// TIA Portal V18 export
// export: Created 2026-01-09T11:31:54.3850951Z, ExportSetting WithDefaults, DisplayName Totally Integrated Automation Portal, DisplayVersion V18 Update 5, DisplayName TIA Portal Openness, DisplayVersion V18 Update 5, DisplayName TIA Portal Teamcenter Gateway, DisplayVersion V18, DisplayName TIA Portal Version Control Interface, DisplayVersion V18, DisplayName SINAMICS Startdrive Advanced, DisplayVersion V18 SP2 Update 1, DisplayName SINAMICS Startdrive G110M, G120, G120C, G120D, G120P, G115D, DisplayVersion V18 SP2 Update 1, DisplayName SINAMICS Startdrive G130, G150, S120, S150, SINAMICS MV, S210, G220, S200, DisplayVersion V18 SP2 Update 1, DisplayName STEP 7 Professional, DisplayVersion V18 Update 5, DisplayName STEP 7 Safety, DisplayVersion V18, DisplayName WinCC Professional, DisplayVersion V18 Update 5
TagTable "ST350_CylinderV2"
  STxxxCylinder001 : fpCylinder V 0.0.19  (%DB1020.DBX0.0, CPU S71500-2PN_TP700, 1 s)
    TagStructureMember "InWP"  LogicalAddress=%DB1020.DBX0.3
    TagStructureMember "InHP"  LogicalAddress=%DB1020.DBX0.4
    TagStructureMember "ValveType"  LogicalAddress=%DB1020.DBX0.5
    TagStructureMember "ManualToWP"  LogicalAddress=%DB1020.DBX6.0
    TagStructureMember "ManualToHP"  LogicalAddress=%DB1020.DBX6.1
    TagStructureMember "GoWorkTime"  LogicalAddress=%DB1020.DBW8
    TagStructureMember "GoHomeTime"  LogicalAddress=%DB1020.DBW10
    TagStructureMember "oGoWP"  LogicalAddress=%DB1020.DBX20.0
    TagStructureMember "oGoHP"  LogicalAddress=%DB1020.DBX20.1
    TagStructureMember "oGoWPBTActive"  LogicalAddress=%DB1020.DBX20.2
    TagStructureMember "oGoHPBTActive"  LogicalAddress=%DB1020.DBX20.3
    TagStructureMember "CylinderNo"  LogicalAddress=%DB1020.DBB21
  STxxxCylinder002 : fpCylinder V 0.0.19  (%DB1020.DBX22.0, CPU S71500-2PN_TP700, 1 s)
    TagStructureMember "InWP"  LogicalAddress=%DB1020.DBX22.3
    TagStructureMember "InHP"  LogicalAddress=%DB1020.DBX22.4
    TagStructureMember "ValveType"  LogicalAddress=%DB1020.DBX22.5
    TagStructureMember "ManualToWP"  LogicalAddress=%DB1020.DBX28.0
    TagStructureMember "ManualToHP"  LogicalAddress=%DB1020.DBX28.1
    TagStructureMember "GoWorkTime"  LogicalAddress=%DB1020.DBW30
    TagStructureMember "GoHomeTime"  LogicalAddress=%DB1020.DBW32
    TagStructureMember "oGoWP"  LogicalAddress=%DB1020.DBX42.0
    TagStructureMember "oGoHP"  LogicalAddress=%DB1020.DBX42.1
    TagStructureMember "oGoWPBTActive"  LogicalAddress=%DB1020.DBX42.2
    TagStructureMember "oGoHPBTActive"  LogicalAddress=%DB1020.DBX42.3
    TagStructureMember "CylinderNo"  LogicalAddress=%DB1020.DBB43
  STxxxCylinder003 : fpCylinder V 0.0.19  (%DB1020.DBX44.0, CPU S71500-2PN_TP700, 1 s)
    TagStructureMember "InWP"  LogicalAddress=%DB1020.DBX44.3
    TagStructureMember "InHP"  LogicalAddress=%DB1020.DBX44.4
    TagStructureMember "ValveType"  LogicalAddress=%DB1020.DBX44.5
    TagStructureMember "ManualToWP"  LogicalAddress=%DB1020.DBX50.0
    TagStructureMember "ManualToHP"  LogicalAddress=%DB1020.DBX50.1
    TagStructureMember "GoWorkTime"  LogicalAddress=%DB1020.DBW52
    TagStructureMember "GoHomeTime"  LogicalAddress=%DB1020.DBW54
    TagStructureMember "oGoWP"  LogicalAddress=%DB1020.DBX64.0
    TagStructureMember "oGoHP"  LogicalAddress=%DB1020.DBX64.1
    TagStructureMember "oGoWPBTActive"  LogicalAddress=%DB1020.DBX64.2
    TagStructureMember "oGoHPBTActive"  LogicalAddress=%DB1020.DBX64.3
    TagStructureMember "CylinderNo"  LogicalAddress=%DB1020.DBB65
  STxxxCylinder004 : fpCylinder V 0.0.19  (%DB1020.DBX66.0, CPU S71500-2PN_TP700, 1 s)
    TagStructureMember "InWP"  LogicalAddress=%DB1020.DBX66.3
    TagStructureMember "InHP"  LogicalAddress=%DB1020.DBX66.4
    TagStructureMember "ValveType"  LogicalAddress=%DB1020.DBX66.5
    TagStructureMember "ManualToWP"  LogicalAddress=%DB1020.DBX72.0
    TagStructureMember "ManualToHP"  LogicalAddress=%DB1020.DBX72.1
    TagStructureMember "GoWorkTime"  LogicalAddress=%DB1020.DBW74
    TagStructureMember "GoHomeTime"  LogicalAddress=%DB1020.DBW76
    TagStructureMember "oGoWP"  LogicalAddress=%DB1020.DBX86.0
    TagStructureMember "oGoHP"  LogicalAddress=%DB1020.DBX86.1
    TagStructureMember "oGoWPBTActive"  LogicalAddress=%DB1020.DBX86.2
    TagStructureMember "oGoHPBTActive"  LogicalAddress=%DB1020.DBX86.3
    TagStructureMember "CylinderNo"  LogicalAddress=%DB1020.DBB87
  STxxxCylinder005 : fpCylinder V 0.0.19  (%DB1020.DBX88.0, CPU S71500-2PN_TP700, 1 s)
    TagStructureMember "InWP"  LogicalAddress=%DB1020.DBX88.3
    TagStructureMember "InHP"  LogicalAddress=%DB1020.DBX88.4
    TagStructureMember "ValveType"  LogicalAddress=%DB1020.DBX88.5
    TagStructureMember "ManualToWP"  LogicalAddress=%DB1020.DBX94.0
    TagStructureMember "ManualToHP"  LogicalAddress=%DB1020.DBX94.1
    TagStructureMember "GoWorkTime"  LogicalAddress=%DB1020.DBW96
    TagStructureMember "GoHomeTime"  LogicalAddress=%DB1020.DBW98
    TagStructureMember "oGoWP"  LogicalAddress=%DB1020.DBX108.0
    TagStructureMember "oGoHP"  LogicalAddress=%DB1020.DBX108.1
    TagStructureMember "oGoWPBTActive"  LogicalAddress=%DB1020.DBX108.2
    TagStructureMember "oGoHPBTActive"  LogicalAddress=%DB1020.DBX108.3
    TagStructureMember "CylinderNo"  LogicalAddress=%DB1020.DBB109
  STxxxCylinder006 : fpCylinder V 0.0.19  (%DB1020.DBX110.0, CPU S71500-2PN_TP700, 1 s)
    TagStructureMember "InWP"  LogicalAddress=%DB1020.DBX110.3
    TagStructureMember "InHP"  LogicalAddress=%DB1020.DBX110.4
    TagStructureMember "ValveType"  LogicalAddress=%DB1020.DBX110.5
    TagStructureMember "ManualToWP"  LogicalAddress=%DB1020.DBX116.0
    TagStructureMember "ManualToHP"  LogicalAddress=%DB1020.DBX116.1
    TagStructureMember "GoWorkTime"  LogicalAddress=%DB1020.DBW118
    TagStructureMember "GoHomeTime"  LogicalAddress=%DB1020.DBW120
    TagStructureMember "oGoWP"  LogicalAddress=%DB1020.DBX130.0
    TagStructureMember "oGoHP"  LogicalAddress=%DB1020.DBX130.1
    TagStructureMember "oGoWPBTActive"  LogicalAddress=%DB1020.DBX130.2
    TagStructureMember "oGoHPBTActive"  LogicalAddress=%DB1020.DBX130.3
    TagStructureMember "CylinderNo"  LogicalAddress=%DB1020.DBB131
  STxxxCylinder007 : fpCylinder V 0.0.19  (%DB1020.DBX132.0, CPU S71500-2PN_TP700, 1 s)
    TagStructureMember "InWP"  LogicalAddress=%DB1020.DBX132.3
    TagStructureMember "InHP"  LogicalAddress=%DB1020.DBX132.4
    TagStructureMember "ValveType"  LogicalAddress=%DB1020.DBX132.5
    TagStructureMember "ManualToWP"  LogicalAddress=%DB1020.DBX138.0
    TagStructureMember "ManualToHP"  LogicalAddress=%DB1020.DBX138.1
    TagStructureMember "GoWorkTime"  LogicalAddress=%DB1020.DBW140
    TagStructureMember "GoHomeTime"  LogicalAddress=%DB1020.DBW142
    TagStructureMember "oGoWP"  LogicalAddress=%DB1020.DBX152.0
    TagStructureMember "oGoHP"  LogicalAddress=%DB1020.DBX152.1
    TagStructureMember "oGoWPBTActive"  LogicalAddress=%DB1020.DBX152.2
    TagStructureMember "oGoHPBTActive"  LogicalAddress=%DB1020.DBX152.3
    TagStructureMember "CylinderNo"  LogicalAddress=%DB1020.DBB153
  STxxxCylinder008 : fpCylinder V 0.0.19  (%DB1020.DBX154.0, CPU S71500-2PN_TP700, 1 s)
    TagStructureMember "InWP"  LogicalAddress=%DB1020.DBX154.3
    TagStructureMember "InHP"  LogicalAddress=%DB1020.DBX154.4
    TagStructureMember "ValveType"  LogicalAddress=%DB1020.DBX154.5
    TagStructureMember "ManualToWP"  LogicalAddress=%DB1020.DBX160.0
    TagStructureMember "ManualToHP"  LogicalAddress=%DB1020.DBX160.1
    TagStructureMember "GoWorkTime"  LogicalAddress=%DB1020.DBW162
    TagStructureMember "GoHomeTime"  LogicalAddress=%DB1020.DBW164
    TagStructureMember "oGoWP"  LogicalAddress=%DB1020.DBX174.0
    TagStructureMember "oGoHP"  LogicalAddress=%DB1020.DBX174.1
    TagStructureMember "oGoWPBTActive"  LogicalAddress=%DB1020.DBX174.2
    TagStructureMember "oGoHPBTActive"  LogicalAddress=%DB1020.DBX174.3
    TagStructureMember "CylinderNo"  LogicalAddress=%DB1020.DBB175
  STxxxCylinder009 : fpCylinder V 0.0.19  (%DB1020.DBX176.0, CPU S71500-2PN_TP700, 1 s)
    TagStructureMember "InWP"  LogicalAddress=%DB1020.DBX176.3
    TagStructureMember "InHP"  LogicalAddress=%DB1020.DBX176.4
    TagStructureMember "ValveType"  LogicalAddress=%DB1020.DBX176.5
    TagStructureMember "ManualToWP"  LogicalAddress=%DB1020.DBX182.0
    TagStructureMember "ManualToHP"  LogicalAddress=%DB1020.DBX182.1
    TagStructureMember "GoWorkTime"  LogicalAddress=%DB1020.DBW184
    TagStructureMember "GoHomeTime"  LogicalAddress=%DB1020.DBW186
    TagStructureMember "oGoWP"  LogicalAddress=%DB1020.DBX196.0
    TagStructureMember "oGoHP"  LogicalAddress=%DB1020.DBX196.1
    TagStructureMember "oGoWPBTActive"  LogicalAddress=%DB1020.DBX196.2
    TagStructureMember "oGoHPBTActive"  LogicalAddress=%DB1020.DBX196.3
    TagStructureMember "CylinderNo"  LogicalAddress=%DB1020.DBB197
  STxxxCylinder010 : fpCylinder V 0.0.19  (%DB1020.DBX198.0, CPU S71500-2PN_TP700, 1 s)
    TagStructureMember "InWP"  LogicalAddress=%DB1020.DBX198.3
    TagStructureMember "InHP"  LogicalAddress=%DB1020.DBX198.4
    TagStructureMember "ValveType"  LogicalAddress=%DB1020.DBX198.5
    TagStructureMember "ManualToWP"  LogicalAddress=%DB1020.DBX204.0
    TagStructureMember "ManualToHP"  LogicalAddress=%DB1020.DBX204.1
    TagStructureMember "GoWorkTime"  LogicalAddress=%DB1020.DBW206
    TagStructureMember "GoHomeTime"  LogicalAddress=%DB1020.DBW208
    TagStructureMember "oGoWP"  LogicalAddress=%DB1020.DBX218.0
    TagStructureMember "oGoHP"  LogicalAddress=%DB1020.DBX218.1
    TagStructureMember "oGoWPBTActive"  LogicalAddress=%DB1020.DBX218.2
    TagStructureMember "oGoHPBTActive"  LogicalAddress=%DB1020.DBX218.3
    TagStructureMember "CylinderNo"  LogicalAddress=%DB1020.DBB219
  STxxxCylinder011 : fpCylinder V 0.0.19  (%DB1020.DBX220.0, CPU S71500-2PN_TP700, 1 s)
    TagStructureMember "InWP"  LogicalAddress=%DB1020.DBX220.3
    TagStructureMember "InHP"  LogicalAddress=%DB1020.DBX220.4
    TagStructureMember "ValveType"  LogicalAddress=%DB1020.DBX220.5
    TagStructureMember "ManualToWP"  LogicalAddress=%DB1020.DBX226.0
    TagStructureMember "ManualToHP"  LogicalAddress=%DB1020.DBX226.1
    TagStructureMember "GoWorkTime"  LogicalAddress=%DB1020.DBW228
    TagStructureMember "GoHomeTime"  LogicalAddress=%DB1020.DBW230
    TagStructureMember "oGoWP"  LogicalAddress=%DB1020.DBX240.0
    TagStructureMember "oGoHP"  LogicalAddress=%DB1020.DBX240.1
    TagStructureMember "oGoWPBTActive"  LogicalAddress=%DB1020.DBX240.2
    TagStructureMember "oGoHPBTActive"  LogicalAddress=%DB1020.DBX240.3
    TagStructureMember "CylinderNo"  LogicalAddress=%DB1020.DBB241
  STxxxCylinder012 : fpCylinder V 0.0.19  (%DB1020.DBX242.0, CPU S71500-2PN_TP700, 1 s)
    TagStructureMember "InWP"  LogicalAddress=%DB1020.DBX242.3
    TagStructureMember "InHP"  LogicalAddress=%DB1020.DBX242.4
    TagStructureMember "ValveType"  LogicalAddress=%DB1020.DBX242.5
    TagStructureMember "ManualToWP"  LogicalAddress=%DB1020.DBX248.0
    TagStructureMember "ManualToHP"  LogicalAddress=%DB1020.DBX248.1
    TagStructureMember "GoWorkTime"  LogicalAddress=%DB1020.DBW250
    TagStructureMember "GoHomeTime"  LogicalAddress=%DB1020.DBW252
    TagStructureMember "oGoWP"  LogicalAddress=%DB1020.DBX262.0
    TagStructureMember "oGoHP"  LogicalAddress=%DB1020.DBX262.1
    TagStructureMember "oGoWPBTActive"  LogicalAddress=%DB1020.DBX262.2
    TagStructureMember "oGoHPBTActive"  LogicalAddress=%DB1020.DBX262.3
    TagStructureMember "CylinderNo"  LogicalAddress=%DB1020.DBB263
  STxxxCylinder013 : fpCylinder V 0.0.19  (%DB1020.DBX264.0, CPU S71500-2PN_TP700, 1 s)
    TagStructureMember "InWP"  LogicalAddress=%DB1020.DBX264.3
    TagStructureMember "InHP"  LogicalAddress=%DB1020.DBX264.4
    TagStructureMember "ValveType"  LogicalAddress=%DB1020.DBX264.5
    TagStructureMember "ManualToWP"  LogicalAddress=%DB1020.DBX270.0
    TagStructureMember "ManualToHP"  LogicalAddress=%DB1020.DBX270.1
    TagStructureMember "GoWorkTime"  LogicalAddress=%DB1020.DBW272
    TagStructureMember "GoHomeTime"  LogicalAddress=%DB1020.DBW274
    TagStructureMember "oGoWP"  LogicalAddress=%DB1020.DBX284.0
    TagStructureMember "oGoHP"  LogicalAddress=%DB1020.DBX284.1
    TagStructureMember "oGoWPBTActive"  LogicalAddress=%DB1020.DBX284.2
    TagStructureMember "oGoHPBTActive"  LogicalAddress=%DB1020.DBX284.3
    TagStructureMember "CylinderNo"  LogicalAddress=%DB1020.DBB285
  STxxxCylinder014 : fpCylinder V 0.0.19  (%DB1020.DBX286.0, CPU S71500-2PN_TP700, 1 s)
    TagStructureMember "InWP"  LogicalAddress=%DB1020.DBX286.3
    TagStructureMember "InHP"  LogicalAddress=%DB1020.DBX286.4
    TagStructureMember "ValveType"  LogicalAddress=%DB1020.DBX286.5
    TagStructureMember "ManualToWP"  LogicalAddress=%DB1020.DBX292.0
    TagStructureMember "ManualToHP"  LogicalAddress=%DB1020.DBX292.1
    TagStructureMember "GoWorkTime"  LogicalAddress=%DB1020.DBW294
    TagStructureMember "GoHomeTime"  LogicalAddress=%DB1020.DBW296
    TagStructureMember "oGoWP"  LogicalAddress=%DB1020.DBX306.0
    TagStructureMember "oGoHP"  LogicalAddress=%DB1020.DBX306.1
    TagStructureMember "oGoWPBTActive"  LogicalAddress=%DB1020.DBX306.2
    TagStructureMember "oGoHPBTActive"  LogicalAddress=%DB1020.DBX306.3
    TagStructureMember "CylinderNo"  LogicalAddress=%DB1020.DBB307
  STxxxCylinder015 : fpCylinder V 0.0.19  (%DB1020.DBX308.0, CPU S71500-2PN_TP700, 1 s)
    TagStructureMember "InWP"  LogicalAddress=%DB1020.DBX308.3
    TagStructureMember "InHP"  LogicalAddress=%DB1020.DBX308.4
    TagStructureMember "ValveType"  LogicalAddress=%DB1020.DBX308.5
    TagStructureMember "ManualToWP"  LogicalAddress=%DB1020.DBX314.0
    TagStructureMember "ManualToHP"  LogicalAddress=%DB1020.DBX314.1
    TagStructureMember "GoWorkTime"  LogicalAddress=%DB1020.DBW316
    TagStructureMember "GoHomeTime"  LogicalAddress=%DB1020.DBW318
    TagStructureMember "oGoWP"  LogicalAddress=%DB1020.DBX328.0
    TagStructureMember "oGoHP"  LogicalAddress=%DB1020.DBX328.1
    TagStructureMember "oGoWPBTActive"  LogicalAddress=%DB1020.DBX328.2
    TagStructureMember "oGoHPBTActive"  LogicalAddress=%DB1020.DBX328.3
    TagStructureMember "CylinderNo"  LogicalAddress=%DB1020.DBB329
  STxxxCylinder016 : fpCylinder V 0.0.19  (%DB1020.DBX330.0, CPU S71500-2PN_TP700, 1 s)
    TagStructureMember "InWP"  LogicalAddress=%DB1020.DBX330.3
    TagStructureMember "InHP"  LogicalAddress=%DB1020.DBX330.4
    TagStructureMember "ValveType"  LogicalAddress=%DB1020.DBX330.5
    TagStructureMember "ManualToWP"  LogicalAddress=%DB1020.DBX336.0
    TagStructureMember "ManualToHP"  LogicalAddress=%DB1020.DBX336.1
    TagStructureMember "GoWorkTime"  LogicalAddress=%DB1020.DBW338
    TagStructureMember "GoHomeTime"  LogicalAddress=%DB1020.DBW340
    TagStructureMember "oGoWP"  LogicalAddress=%DB1020.DBX350.0
    TagStructureMember "oGoHP"  LogicalAddress=%DB1020.DBX350.1
    TagStructureMember "oGoWPBTActive"  LogicalAddress=%DB1020.DBX350.2
    TagStructureMember "oGoHPBTActive"  LogicalAddress=%DB1020.DBX350.3
    TagStructureMember "CylinderNo"  LogicalAddress=%DB1020.DBB351
  STxxxCylinder017 : fpCylinder V 0.0.19  (%DB1020.DBX352.0, CPU S71500-2PN_TP700, 1 s)
    TagStructureMember "InWP"  LogicalAddress=%DB1020.DBX352.3
    TagStructureMember "InHP"  LogicalAddress=%DB1020.DBX352.4
    TagStructureMember "ValveType"  LogicalAddress=%DB1020.DBX352.5
    TagStructureMember "ManualToWP"  LogicalAddress=%DB1020.DBX358.0
    TagStructureMember "ManualToHP"  LogicalAddress=%DB1020.DBX358.1
    TagStructureMember "GoWorkTime"  LogicalAddress=%DB1020.DBW360
    TagStructureMember "GoHomeTime"  LogicalAddress=%DB1020.DBW362
    TagStructureMember "oGoWP"  LogicalAddress=%DB1020.DBX372.0
    TagStructureMember "oGoHP"  LogicalAddress=%DB1020.DBX372.1
    TagStructureMember "oGoWPBTActive"  LogicalAddress=%DB1020.DBX372.2
    TagStructureMember "oGoHPBTActive"  LogicalAddress=%DB1020.DBX372.3
    TagStructureMember "CylinderNo"  LogicalAddress=%DB1020.DBB373
  STxxxCylinder018 : fpCylinder V 0.0.19  (%DB1020.DBX374.0, CPU S71500-2PN_TP700, 1 s)
    TagStructureMember "InWP"  LogicalAddress=%DB1020.DBX374.3
    TagStructureMember "InHP"  LogicalAddress=%DB1020.DBX374.4
    TagStructureMember "ValveType"  LogicalAddress=%DB1020.DBX374.5
    TagStructureMember "ManualToWP"  LogicalAddress=%DB1020.DBX380.0
    TagStructureMember "ManualToHP"  LogicalAddress=%DB1020.DBX380.1
    TagStructureMember "GoWorkTime"  LogicalAddress=%DB1020.DBW382
    TagStructureMember "GoHomeTime"  LogicalAddress=%DB1020.DBW384
    TagStructureMember "oGoWP"  LogicalAddress=%DB1020.DBX394.0
    TagStructureMember "oGoHP"  LogicalAddress=%DB1020.DBX394.1
    TagStructureMember "oGoWPBTActive"  LogicalAddress=%DB1020.DBX394.2
    TagStructureMember "oGoHPBTActive"  LogicalAddress=%DB1020.DBX394.3
    TagStructureMember "CylinderNo"  LogicalAddress=%DB1020.DBB395
  STxxxCylinder019 : fpCylinder V 0.0.19  (%DB1020.DBX396.0, CPU S71500-2PN_TP700, 1 s)
    TagStructureMember "InWP"  LogicalAddress=%DB1020.DBX396.3
    TagStructureMember "InHP"  LogicalAddress=%DB1020.DBX396.4
    TagStructureMember "ValveType"  LogicalAddress=%DB1020.DBX396.5
    TagStructureMember "ManualToWP"  LogicalAddress=%DB1020.DBX402.0
    TagStructureMember "ManualToHP"  LogicalAddress=%DB1020.DBX402.1
    TagStructureMember "GoWorkTime"  LogicalAddress=%DB1020.DBW404
    TagStructureMember "GoHomeTime"  LogicalAddress=%DB1020.DBW406
    TagStructureMember "oGoWP"  LogicalAddress=%DB1020.DBX416.0
    TagStructureMember "oGoHP"  LogicalAddress=%DB1020.DBX416.1
    TagStructureMember "oGoWPBTActive"  LogicalAddress=%DB1020.DBX416.2
    TagStructureMember "oGoHPBTActive"  LogicalAddress=%DB1020.DBX416.3
    TagStructureMember "CylinderNo"  LogicalAddress=%DB1020.DBB417
  STxxxCylinder020 : fpCylinder V 0.0.19  (%DB1020.DBX418.0, CPU S71500-2PN_TP700, 1 s)
    TagStructureMember "InWP"  LogicalAddress=%DB1020.DBX418.3
    TagStructureMember "InHP"  LogicalAddress=%DB1020.DBX418.4
    TagStructureMember "ValveType"  LogicalAddress=%DB1020.DBX418.5
    TagStructureMember "ManualToWP"  LogicalAddress=%DB1020.DBX424.0
    TagStructureMember "ManualToHP"  LogicalAddress=%DB1020.DBX424.1
    TagStructureMember "GoWorkTime"  LogicalAddress=%DB1020.DBW426
    TagStructureMember "GoHomeTime"  LogicalAddress=%DB1020.DBW428
    TagStructureMember "oGoWP"  LogicalAddress=%DB1020.DBX438.0
    TagStructureMember "oGoHP"  LogicalAddress=%DB1020.DBX438.1
    TagStructureMember "oGoWPBTActive"  LogicalAddress=%DB1020.DBX438.2
    TagStructureMember "oGoHPBTActive"  LogicalAddress=%DB1020.DBX438.3
    TagStructureMember "CylinderNo"  LogicalAddress=%DB1020.DBB439
  STxxxCylinder021 : fpCylinder V 0.0.19  (%DB1020.DBX440.0, CPU S71500-2PN_TP700, 1 s)
    TagStructureMember "InWP"  LogicalAddress=%DB1020.DBX440.3
    TagStructureMember "InHP"  LogicalAddress=%DB1020.DBX440.4
    TagStructureMember "ValveType"  LogicalAddress=%DB1020.DBX440.5
    TagStructureMember "ManualToWP"  LogicalAddress=%DB1020.DBX446.0
    TagStructureMember "ManualToHP"  LogicalAddress=%DB1020.DBX446.1
    TagStructureMember "GoWorkTime"  LogicalAddress=%DB1020.DBW448
    TagStructureMember "GoHomeTime"  LogicalAddress=%DB1020.DBW450
    TagStructureMember "oGoWP"  LogicalAddress=%DB1020.DBX460.0
    TagStructureMember "oGoHP"  LogicalAddress=%DB1020.DBX460.1
    TagStructureMember "oGoWPBTActive"  LogicalAddress=%DB1020.DBX460.2
    TagStructureMember "oGoHPBTActive"  LogicalAddress=%DB1020.DBX460.3
    TagStructureMember "CylinderNo"  LogicalAddress=%DB1020.DBB461
  STxxxCylinder022 : fpCylinder V 0.0.19  (%DB1020.DBX462.0, CPU S71500-2PN_TP700, 1 s)
    TagStructureMember "InWP"  LogicalAddress=%DB1020.DBX462.3
    TagStructureMember "InHP"  LogicalAddress=%DB1020.DBX462.4
    TagStructureMember "ValveType"  LogicalAddress=%DB1020.DBX462.5
    TagStructureMember "ManualToWP"  LogicalAddress=%DB1020.DBX468.0
    TagStructureMember "ManualToHP"  LogicalAddress=%DB1020.DBX468.1
    TagStructureMember "GoWorkTime"  LogicalAddress=%DB1020.DBW470
    TagStructureMember "GoHomeTime"  LogicalAddress=%DB1020.DBW472
    TagStructureMember "oGoWP"  LogicalAddress=%DB1020.DBX482.0
    TagStructureMember "oGoHP"  LogicalAddress=%DB1020.DBX482.1
    TagStructureMember "oGoWPBTActive"  LogicalAddress=%DB1020.DBX482.2
    TagStructureMember "oGoHPBTActive"  LogicalAddress=%DB1020.DBX482.3
    TagStructureMember "CylinderNo"  LogicalAddress=%DB1020.DBB483
  STxxxCylinder023 : fpCylinder V 0.0.19  (%DB1020.DBX484.0, CPU S71500-2PN_TP700, 1 s)
    TagStructureMember "InWP"  LogicalAddress=%DB1020.DBX484.3
    TagStructureMember "InHP"  LogicalAddress=%DB1020.DBX484.4
    TagStructureMember "ValveType"  LogicalAddress=%DB1020.DBX484.5
    TagStructureMember "ManualToWP"  LogicalAddress=%DB1020.DBX490.0
    TagStructureMember "ManualToHP"  LogicalAddress=%DB1020.DBX490.1
    TagStructureMember "GoWorkTime"  LogicalAddress=%DB1020.DBW492
    TagStructureMember "GoHomeTime"  LogicalAddress=%DB1020.DBW494
    TagStructureMember "oGoWP"  LogicalAddress=%DB1020.DBX504.0
    TagStructureMember "oGoHP"  LogicalAddress=%DB1020.DBX504.1
    TagStructureMember "oGoWPBTActive"  LogicalAddress=%DB1020.DBX504.2
    TagStructureMember "oGoHPBTActive"  LogicalAddress=%DB1020.DBX504.3
    TagStructureMember "CylinderNo"  LogicalAddress=%DB1020.DBB505
  STxxxCylinder024 : fpCylinder V 0.0.19  (%DB1020.DBX506.0, CPU S71500-2PN_TP700, 1 s)
    TagStructureMember "InWP"  LogicalAddress=%DB1020.DBX506.3
    TagStructureMember "InHP"  LogicalAddress=%DB1020.DBX506.4
    TagStructureMember "ValveType"  LogicalAddress=%DB1020.DBX506.5
    TagStructureMember "ManualToWP"  LogicalAddress=%DB1020.DBX512.0
    TagStructureMember "ManualToHP"  LogicalAddress=%DB1020.DBX512.1
    TagStructureMember "GoWorkTime"  LogicalAddress=%DB1020.DBW514
    TagStructureMember "GoHomeTime"  LogicalAddress=%DB1020.DBW516
    TagStructureMember "oGoWP"  LogicalAddress=%DB1020.DBX526.0
    TagStructureMember "oGoHP"  LogicalAddress=%DB1020.DBX526.1
    TagStructureMember "oGoWPBTActive"  LogicalAddress=%DB1020.DBX526.2
    TagStructureMember "oGoHPBTActive"  LogicalAddress=%DB1020.DBX526.3
    TagStructureMember "CylinderNo"  LogicalAddress=%DB1020.DBB527
  STxxxCylinder025 : fpCylinder V 0.0.19  (%DB1020.DBX528.0, CPU S71500-2PN_TP700, 1 s)
    TagStructureMember "InWP"  LogicalAddress=%DB1020.DBX528.3
    TagStructureMember "InHP"  LogicalAddress=%DB1020.DBX528.4
    TagStructureMember "ValveType"  LogicalAddress=%DB1020.DBX528.5
    TagStructureMember "ManualToWP"  LogicalAddress=%DB1020.DBX534.0
    TagStructureMember "ManualToHP"  LogicalAddress=%DB1020.DBX534.1
    TagStructureMember "GoWorkTime"  LogicalAddress=%DB1020.DBW536
    TagStructureMember "GoHomeTime"  LogicalAddress=%DB1020.DBW538
    TagStructureMember "oGoWP"  LogicalAddress=%DB1020.DBX548.0
    TagStructureMember "oGoHP"  LogicalAddress=%DB1020.DBX548.1
    TagStructureMember "oGoWPBTActive"  LogicalAddress=%DB1020.DBX548.2
    TagStructureMember "oGoHPBTActive"  LogicalAddress=%DB1020.DBX548.3
    TagStructureMember "CylinderNo"  LogicalAddress=%DB1020.DBB549
  STxxxCylinder026 : fpCylinder V 0.0.19  (%DB1020.DBX550.0, CPU S71500-2PN_TP700, 1 s)
    TagStructureMember "InWP"  LogicalAddress=%DB1020.DBX550.3
    TagStructureMember "InHP"  LogicalAddress=%DB1020.DBX550.4
    TagStructureMember "ValveType"  LogicalAddress=%DB1020.DBX550.5
    TagStructureMember "ManualToWP"  LogicalAddress=%DB1020.DBX556.0
    TagStructureMember "ManualToHP"  LogicalAddress=%DB1020.DBX556.1
    TagStructureMember "GoWorkTime"  LogicalAddress=%DB1020.DBW558
    TagStructureMember "GoHomeTime"  LogicalAddress=%DB1020.DBW560
    TagStructureMember "oGoWP"  LogicalAddress=%DB1020.DBX570.0
    TagStructureMember "oGoHP"  LogicalAddress=%DB1020.DBX570.1
    TagStructureMember "oGoWPBTActive"  LogicalAddress=%DB1020.DBX570.2
    TagStructureMember "oGoHPBTActive"  LogicalAddress=%DB1020.DBX570.3
    TagStructureMember "CylinderNo"  LogicalAddress=%DB1020.DBB571
  STxxxCylinder027 : fpCylinder V 0.0.19  (%DB1020.DBX572.0, CPU S71500-2PN_TP700, 1 s)
    TagStructureMember "InWP"  LogicalAddress=%DB1020.DBX572.3
    TagStructureMember "InHP"  LogicalAddress=%DB1020.DBX572.4
    TagStructureMember "ValveType"  LogicalAddress=%DB1020.DBX572.5
    TagStructureMember "ManualToWP"  LogicalAddress=%DB1020.DBX578.0
    TagStructureMember "ManualToHP"  LogicalAddress=%DB1020.DBX578.1
    TagStructureMember "GoWorkTime"  LogicalAddress=%DB1020.DBW580
    TagStructureMember "GoHomeTime"  LogicalAddress=%DB1020.DBW582
    TagStructureMember "oGoWP"  LogicalAddress=%DB1020.DBX592.0
    TagStructureMember "oGoHP"  LogicalAddress=%DB1020.DBX592.1
    TagStructureMember "oGoWPBTActive"  LogicalAddress=%DB1020.DBX592.2
    TagStructureMember "oGoHPBTActive"  LogicalAddress=%DB1020.DBX592.3
    TagStructureMember "CylinderNo"  LogicalAddress=%DB1020.DBB593
  STxxxCylinder028 : fpCylinder V 0.0.19  (%DB1020.DBX594.0, CPU S71500-2PN_TP700, 1 s)
    TagStructureMember "InWP"  LogicalAddress=%DB1020.DBX594.3
    TagStructureMember "InHP"  LogicalAddress=%DB1020.DBX594.4
    TagStructureMember "ValveType"  LogicalAddress=%DB1020.DBX594.5
    TagStructureMember "ManualToWP"  LogicalAddress=%DB1020.DBX600.0
    TagStructureMember "ManualToHP"  LogicalAddress=%DB1020.DBX600.1
    TagStructureMember "GoWorkTime"  LogicalAddress=%DB1020.DBW602
    TagStructureMember "GoHomeTime"  LogicalAddress=%DB1020.DBW604
    TagStructureMember "oGoWP"  LogicalAddress=%DB1020.DBX614.0
    TagStructureMember "oGoHP"  LogicalAddress=%DB1020.DBX614.1
    TagStructureMember "oGoWPBTActive"  LogicalAddress=%DB1020.DBX614.2
    TagStructureMember "oGoHPBTActive"  LogicalAddress=%DB1020.DBX614.3
    TagStructureMember "CylinderNo"  LogicalAddress=%DB1020.DBB615
  STxxxCylinder029 : fpCylinder V 0.0.19  (%DB1020.DBX616.0, CPU S71500-2PN_TP700, 1 s)
    TagStructureMember "InWP"  LogicalAddress=%DB1020.DBX616.3
    TagStructureMember "InHP"  LogicalAddress=%DB1020.DBX616.4
    TagStructureMember "ValveType"  LogicalAddress=%DB1020.DBX616.5
    TagStructureMember "ManualToWP"  LogicalAddress=%DB1020.DBX622.0
    TagStructureMember "ManualToHP"  LogicalAddress=%DB1020.DBX622.1
    TagStructureMember "GoWorkTime"  LogicalAddress=%DB1020.DBW624
    TagStructureMember "GoHomeTime"  LogicalAddress=%DB1020.DBW626
    TagStructureMember "oGoWP"  LogicalAddress=%DB1020.DBX636.0
    TagStructureMember "oGoHP"  LogicalAddress=%DB1020.DBX636.1
    TagStructureMember "oGoWPBTActive"  LogicalAddress=%DB1020.DBX636.2
    TagStructureMember "oGoHPBTActive"  LogicalAddress=%DB1020.DBX636.3
    TagStructureMember "CylinderNo"  LogicalAddress=%DB1020.DBB637
  STxxxCylinder030 : fpCylinder V 0.0.19  (%DB1020.DBX638.0, CPU S71500-2PN_TP700, 1 s)
    TagStructureMember "InWP"  LogicalAddress=%DB1020.DBX638.3
    TagStructureMember "InHP"  LogicalAddress=%DB1020.DBX638.4
    TagStructureMember "ValveType"  LogicalAddress=%DB1020.DBX638.5
    TagStructureMember "ManualToWP"  LogicalAddress=%DB1020.DBX644.0
    TagStructureMember "ManualToHP"  LogicalAddress=%DB1020.DBX644.1
    TagStructureMember "GoWorkTime"  LogicalAddress=%DB1020.DBW646
    TagStructureMember "GoHomeTime"  LogicalAddress=%DB1020.DBW648
    TagStructureMember "oGoWP"  LogicalAddress=%DB1020.DBX658.0
    TagStructureMember "oGoHP"  LogicalAddress=%DB1020.DBX658.1
    TagStructureMember "oGoWPBTActive"  LogicalAddress=%DB1020.DBX658.2
    TagStructureMember "oGoHPBTActive"  LogicalAddress=%DB1020.DBX658.3
    TagStructureMember "CylinderNo"  LogicalAddress=%DB1020.DBB659
  STxxxCylinder031 : fpCylinder V 0.0.19  (%DB1020.DBX660.0, CPU S71500-2PN_TP700, 1 s)
    TagStructureMember "InWP"  LogicalAddress=%DB1020.DBX660.3
    TagStructureMember "InHP"  LogicalAddress=%DB1020.DBX660.4
    TagStructureMember "ValveType"  LogicalAddress=%DB1020.DBX660.5
    TagStructureMember "ManualToWP"  LogicalAddress=%DB1020.DBX666.0
    TagStructureMember "ManualToHP"  LogicalAddress=%DB1020.DBX666.1
    TagStructureMember "GoWorkTime"  LogicalAddress=%DB1020.DBW668
    TagStructureMember "GoHomeTime"  LogicalAddress=%DB1020.DBW670
    TagStructureMember "oGoWP"  LogicalAddress=%DB1020.DBX680.0
    TagStructureMember "oGoHP"  LogicalAddress=%DB1020.DBX680.1
    TagStructureMember "oGoWPBTActive"  LogicalAddress=%DB1020.DBX680.2
    TagStructureMember "oGoHPBTActive"  LogicalAddress=%DB1020.DBX680.3
    TagStructureMember "CylinderNo"  LogicalAddress=%DB1020.DBB681
  STxxxCylinder032 : fpCylinder V 0.0.19  (%DB1020.DBX682.0, CPU S71500-2PN_TP700, 1 s)
    TagStructureMember "InWP"  LogicalAddress=%DB1020.DBX682.3
    TagStructureMember "InHP"  LogicalAddress=%DB1020.DBX682.4
    TagStructureMember "ValveType"  LogicalAddress=%DB1020.DBX682.5
    TagStructureMember "ManualToWP"  LogicalAddress=%DB1020.DBX688.0
    TagStructureMember "ManualToHP"  LogicalAddress=%DB1020.DBX688.1
    TagStructureMember "GoWorkTime"  LogicalAddress=%DB1020.DBW690
    TagStructureMember "GoHomeTime"  LogicalAddress=%DB1020.DBW692
    TagStructureMember "oGoWP"  LogicalAddress=%DB1020.DBX702.0
    TagStructureMember "oGoHP"  LogicalAddress=%DB1020.DBX702.1
    TagStructureMember "oGoWPBTActive"  LogicalAddress=%DB1020.DBX702.2
    TagStructureMember "oGoHPBTActive"  LogicalAddress=%DB1020.DBX702.3
    TagStructureMember "CylinderNo"  LogicalAddress=%DB1020.DBB703
  STxxxCylinder033 : fpCylinder V 0.0.19  (%DB1020.DBX704.0, CPU S71500-2PN_TP700, 1 s)
    TagStructureMember "InWP"  LogicalAddress=%DB1020.DBX704.3
    TagStructureMember "InHP"  LogicalAddress=%DB1020.DBX704.4
    TagStructureMember "ValveType"  LogicalAddress=%DB1020.DBX704.5
    TagStructureMember "ManualToWP"  LogicalAddress=%DB1020.DBX710.0
    TagStructureMember "ManualToHP"  LogicalAddress=%DB1020.DBX710.1
    TagStructureMember "GoWorkTime"  LogicalAddress=%DB1020.DBW712
    TagStructureMember "GoHomeTime"  LogicalAddress=%DB1020.DBW714
    TagStructureMember "oGoWP"  LogicalAddress=%DB1020.DBX724.0
    TagStructureMember "oGoHP"  LogicalAddress=%DB1020.DBX724.1
    TagStructureMember "oGoWPBTActive"  LogicalAddress=%DB1020.DBX724.2
    TagStructureMember "oGoHPBTActive"  LogicalAddress=%DB1020.DBX724.3
    TagStructureMember "CylinderNo"  LogicalAddress=%DB1020.DBB725
  STxxxCylinder034 : fpCylinder V 0.0.19  (%DB1020.DBX726.0, CPU S71500-2PN_TP700, 1 s)
    TagStructureMember "InWP"  LogicalAddress=%DB1020.DBX726.3
    TagStructureMember "InHP"  LogicalAddress=%DB1020.DBX726.4
    TagStructureMember "ValveType"  LogicalAddress=%DB1020.DBX726.5
    TagStructureMember "ManualToWP"  LogicalAddress=%DB1020.DBX732.0
    TagStructureMember "ManualToHP"  LogicalAddress=%DB1020.DBX732.1
    TagStructureMember "GoWorkTime"  LogicalAddress=%DB1020.DBW734
    TagStructureMember "GoHomeTime"  LogicalAddress=%DB1020.DBW736
    TagStructureMember "oGoWP"  LogicalAddress=%DB1020.DBX746.0
    TagStructureMember "oGoHP"  LogicalAddress=%DB1020.DBX746.1
    TagStructureMember "oGoWPBTActive"  LogicalAddress=%DB1020.DBX746.2
    TagStructureMember "oGoHPBTActive"  LogicalAddress=%DB1020.DBX746.3
    TagStructureMember "CylinderNo"  LogicalAddress=%DB1020.DBB747
  STxxxCylinder035 : fpCylinder V 0.0.19  (%DB1020.DBX748.0, CPU S71500-2PN_TP700, 1 s)
    TagStructureMember "InWP"  LogicalAddress=%DB1020.DBX748.3
    TagStructureMember "InHP"  LogicalAddress=%DB1020.DBX748.4
    TagStructureMember "ValveType"  LogicalAddress=%DB1020.DBX748.5
    TagStructureMember "ManualToWP"  LogicalAddress=%DB1020.DBX754.0
    TagStructureMember "ManualToHP"  LogicalAddress=%DB1020.DBX754.1
    TagStructureMember "GoWorkTime"  LogicalAddress=%DB1020.DBW756
    TagStructureMember "GoHomeTime"  LogicalAddress=%DB1020.DBW758
    TagStructureMember "oGoWP"  LogicalAddress=%DB1020.DBX768.0
    TagStructureMember "oGoHP"  LogicalAddress=%DB1020.DBX768.1
    TagStructureMember "oGoWPBTActive"  LogicalAddress=%DB1020.DBX768.2
    TagStructureMember "oGoHPBTActive"  LogicalAddress=%DB1020.DBX768.3
    TagStructureMember "CylinderNo"  LogicalAddress=%DB1020.DBB769
  STxxxCylinder036 : fpCylinder V 0.0.19  (%DB1020.DBX770.0, CPU S71500-2PN_TP700, 1 s)
    TagStructureMember "InWP"  LogicalAddress=%DB1020.DBX770.3
    TagStructureMember "InHP"  LogicalAddress=%DB1020.DBX770.4
    TagStructureMember "ValveType"  LogicalAddress=%DB1020.DBX770.5
    TagStructureMember "ManualToWP"  LogicalAddress=%DB1020.DBX776.0
    TagStructureMember "ManualToHP"  LogicalAddress=%DB1020.DBX776.1
    TagStructureMember "GoWorkTime"  LogicalAddress=%DB1020.DBW778
    TagStructureMember "GoHomeTime"  LogicalAddress=%DB1020.DBW780
    TagStructureMember "oGoWP"  LogicalAddress=%DB1020.DBX790.0
    TagStructureMember "oGoHP"  LogicalAddress=%DB1020.DBX790.1
    TagStructureMember "oGoWPBTActive"  LogicalAddress=%DB1020.DBX790.2
    TagStructureMember "oGoHPBTActive"  LogicalAddress=%DB1020.DBX790.3
    TagStructureMember "CylinderNo"  LogicalAddress=%DB1020.DBB791
  STxxxCylinder037 : fpCylinder V 0.0.19  (%DB1020.DBX792.0, CPU S71500-2PN_TP700, 1 s)
    TagStructureMember "InWP"  LogicalAddress=%DB1020.DBX792.3
    TagStructureMember "InHP"  LogicalAddress=%DB1020.DBX792.4
    TagStructureMember "ValveType"  LogicalAddress=%DB1020.DBX792.5
    TagStructureMember "ManualToWP"  LogicalAddress=%DB1020.DBX798.0
    TagStructureMember "ManualToHP"  LogicalAddress=%DB1020.DBX798.1
    TagStructureMember "GoWorkTime"  LogicalAddress=%DB1020.DBW800
    TagStructureMember "GoHomeTime"  LogicalAddress=%DB1020.DBW802
    TagStructureMember "oGoWP"  LogicalAddress=%DB1020.DBX812.0
    TagStructureMember "oGoHP"  LogicalAddress=%DB1020.DBX812.1
    TagStructureMember "oGoWPBTActive"  LogicalAddress=%DB1020.DBX812.2
    TagStructureMember "oGoHPBTActive"  LogicalAddress=%DB1020.DBX812.3
    TagStructureMember "CylinderNo"  LogicalAddress=%DB1020.DBB813
  STxxxCylinder038 : fpCylinder V 0.0.19  (%DB1020.DBX814.0, CPU S71500-2PN_TP700, 1 s)
    TagStructureMember "InWP"  LogicalAddress=%DB1020.DBX814.3
    TagStructureMember "InHP"  LogicalAddress=%DB1020.DBX814.4
    TagStructureMember "ValveType"  LogicalAddress=%DB1020.DBX814.5
    TagStructureMember "ManualToWP"  LogicalAddress=%DB1020.DBX820.0
    TagStructureMember "ManualToHP"  LogicalAddress=%DB1020.DBX820.1
    TagStructureMember "GoWorkTime"  LogicalAddress=%DB1020.DBW822
    TagStructureMember "GoHomeTime"  LogicalAddress=%DB1020.DBW824
    TagStructureMember "oGoWP"  LogicalAddress=%DB1020.DBX834.0
    TagStructureMember "oGoHP"  LogicalAddress=%DB1020.DBX834.1
    TagStructureMember "oGoWPBTActive"  LogicalAddress=%DB1020.DBX834.2
    TagStructureMember "oGoHPBTActive"  LogicalAddress=%DB1020.DBX834.3
    TagStructureMember "CylinderNo"  LogicalAddress=%DB1020.DBB835
  STxxxCylinder039 : fpCylinder V 0.0.19  (%DB1020.DBX836.0, CPU S71500-2PN_TP700, 1 s)
    TagStructureMember "InWP"  LogicalAddress=%DB1020.DBX836.3
    TagStructureMember "InHP"  LogicalAddress=%DB1020.DBX836.4
    TagStructureMember "ValveType"  LogicalAddress=%DB1020.DBX836.5
    TagStructureMember "ManualToWP"  LogicalAddress=%DB1020.DBX842.0
    TagStructureMember "ManualToHP"  LogicalAddress=%DB1020.DBX842.1
    TagStructureMember "GoWorkTime"  LogicalAddress=%DB1020.DBW844
    TagStructureMember "GoHomeTime"  LogicalAddress=%DB1020.DBW846
    TagStructureMember "oGoWP"  LogicalAddress=%DB1020.DBX856.0
    TagStructureMember "oGoHP"  LogicalAddress=%DB1020.DBX856.1
    TagStructureMember "oGoWPBTActive"  LogicalAddress=%DB1020.DBX856.2
    TagStructureMember "oGoHPBTActive"  LogicalAddress=%DB1020.DBX856.3
    TagStructureMember "CylinderNo"  LogicalAddress=%DB1020.DBB857
  STxxxCylinder040 : fpCylinder V 0.0.19  (%DB1020.DBX858.0, CPU S71500-2PN_TP700, 1 s)
    TagStructureMember "InWP"  LogicalAddress=%DB1020.DBX858.3
    TagStructureMember "InHP"  LogicalAddress=%DB1020.DBX858.4
    TagStructureMember "ValveType"  LogicalAddress=%DB1020.DBX858.5
    TagStructureMember "ManualToWP"  LogicalAddress=%DB1020.DBX864.0
    TagStructureMember "ManualToHP"  LogicalAddress=%DB1020.DBX864.1
    TagStructureMember "GoWorkTime"  LogicalAddress=%DB1020.DBW866
    TagStructureMember "GoHomeTime"  LogicalAddress=%DB1020.DBW868
    TagStructureMember "oGoWP"  LogicalAddress=%DB1020.DBX878.0
    TagStructureMember "oGoHP"  LogicalAddress=%DB1020.DBX878.1
    TagStructureMember "oGoWPBTActive"  LogicalAddress=%DB1020.DBX878.2
    TagStructureMember "oGoHPBTActive"  LogicalAddress=%DB1020.DBX878.3
    TagStructureMember "CylinderNo"  LogicalAddress=%DB1020.DBB879
  STxxxCylinder041 : fpCylinder V 0.0.19  (%DB1020.DBX880.0, CPU S71500-2PN_TP700, 1 s)
    TagStructureMember "InWP"  LogicalAddress=%DB1020.DBX880.3
    TagStructureMember "InHP"  LogicalAddress=%DB1020.DBX880.4
    TagStructureMember "ValveType"  LogicalAddress=%DB1020.DBX880.5
    TagStructureMember "ManualToWP"  LogicalAddress=%DB1020.DBX886.0
    TagStructureMember "ManualToHP"  LogicalAddress=%DB1020.DBX886.1
    TagStructureMember "GoWorkTime"  LogicalAddress=%DB1020.DBW888
    TagStructureMember "GoHomeTime"  LogicalAddress=%DB1020.DBW890
    TagStructureMember "oGoWP"  LogicalAddress=%DB1020.DBX900.0
    TagStructureMember "oGoHP"  LogicalAddress=%DB1020.DBX900.1
    TagStructureMember "oGoWPBTActive"  LogicalAddress=%DB1020.DBX900.2
    TagStructureMember "oGoHPBTActive"  LogicalAddress=%DB1020.DBX900.3
    TagStructureMember "CylinderNo"  LogicalAddress=%DB1020.DBB901
  STxxxCylinder042 : fpCylinder V 0.0.19  (%DB1020.DBX902.0, CPU S71500-2PN_TP700, 1 s)
    TagStructureMember "InWP"  LogicalAddress=%DB1020.DBX902.3
    TagStructureMember "InHP"  LogicalAddress=%DB1020.DBX902.4
    TagStructureMember "ValveType"  LogicalAddress=%DB1020.DBX902.5
    TagStructureMember "ManualToWP"  LogicalAddress=%DB1020.DBX908.0
    TagStructureMember "ManualToHP"  LogicalAddress=%DB1020.DBX908.1
    TagStructureMember "GoWorkTime"  LogicalAddress=%DB1020.DBW910
    TagStructureMember "GoHomeTime"  LogicalAddress=%DB1020.DBW912
    TagStructureMember "oGoWP"  LogicalAddress=%DB1020.DBX922.0
    TagStructureMember "oGoHP"  LogicalAddress=%DB1020.DBX922.1
    TagStructureMember "oGoWPBTActive"  LogicalAddress=%DB1020.DBX922.2
    TagStructureMember "oGoHPBTActive"  LogicalAddress=%DB1020.DBX922.3
    TagStructureMember "CylinderNo"  LogicalAddress=%DB1020.DBB923
  STxxxCylinder043 : fpCylinder V 0.0.19  (%DB1020.DBX924.0, CPU S71500-2PN_TP700, 1 s)
    TagStructureMember "InWP"  LogicalAddress=%DB1020.DBX924.3
    TagStructureMember "InHP"  LogicalAddress=%DB1020.DBX924.4
    TagStructureMember "ValveType"  LogicalAddress=%DB1020.DBX924.5
    TagStructureMember "ManualToWP"  LogicalAddress=%DB1020.DBX930.0
    TagStructureMember "ManualToHP"  LogicalAddress=%DB1020.DBX930.1
    TagStructureMember "GoWorkTime"  LogicalAddress=%DB1020.DBW932
    TagStructureMember "GoHomeTime"  LogicalAddress=%DB1020.DBW934
    TagStructureMember "oGoWP"  LogicalAddress=%DB1020.DBX944.0
    TagStructureMember "oGoHP"  LogicalAddress=%DB1020.DBX944.1
    TagStructureMember "oGoWPBTActive"  LogicalAddress=%DB1020.DBX944.2
    TagStructureMember "oGoHPBTActive"  LogicalAddress=%DB1020.DBX944.3
    TagStructureMember "CylinderNo"  LogicalAddress=%DB1020.DBB945
  STxxxCylinder044 : fpCylinder V 0.0.19  (%DB1020.DBX946.0, CPU S71500-2PN_TP700, 1 s)
    TagStructureMember "InWP"  LogicalAddress=%DB1020.DBX946.3
    TagStructureMember "InHP"  LogicalAddress=%DB1020.DBX946.4
    TagStructureMember "ValveType"  LogicalAddress=%DB1020.DBX946.5
    TagStructureMember "ManualToWP"  LogicalAddress=%DB1020.DBX952.0
    TagStructureMember "ManualToHP"  LogicalAddress=%DB1020.DBX952.1
    TagStructureMember "GoWorkTime"  LogicalAddress=%DB1020.DBW954
    TagStructureMember "GoHomeTime"  LogicalAddress=%DB1020.DBW956
    TagStructureMember "oGoWP"  LogicalAddress=%DB1020.DBX966.0
    TagStructureMember "oGoHP"  LogicalAddress=%DB1020.DBX966.1
    TagStructureMember "oGoWPBTActive"  LogicalAddress=%DB1020.DBX966.2
    TagStructureMember "oGoHPBTActive"  LogicalAddress=%DB1020.DBX966.3
    TagStructureMember "CylinderNo"  LogicalAddress=%DB1020.DBB967
  STxxxCylinder045 : fpCylinder V 0.0.19  (%DB1020.DBX968.0, CPU S71500-2PN_TP700, 1 s)
    TagStructureMember "InWP"  LogicalAddress=%DB1020.DBX968.3
    TagStructureMember "InHP"  LogicalAddress=%DB1020.DBX968.4
    TagStructureMember "ValveType"  LogicalAddress=%DB1020.DBX968.5
    TagStructureMember "ManualToWP"  LogicalAddress=%DB1020.DBX974.0
    TagStructureMember "ManualToHP"  LogicalAddress=%DB1020.DBX974.1
    TagStructureMember "GoWorkTime"  LogicalAddress=%DB1020.DBW976
    TagStructureMember "GoHomeTime"  LogicalAddress=%DB1020.DBW978
    TagStructureMember "oGoWP"  LogicalAddress=%DB1020.DBX988.0
    TagStructureMember "oGoHP"  LogicalAddress=%DB1020.DBX988.1
    TagStructureMember "oGoWPBTActive"  LogicalAddress=%DB1020.DBX988.2
    TagStructureMember "oGoHPBTActive"  LogicalAddress=%DB1020.DBX988.3
    TagStructureMember "CylinderNo"  LogicalAddress=%DB1020.DBB989
  STxxxCylinder046 : fpCylinder V 0.0.19  (%DB1020.DBX990.0, CPU S71500-2PN_TP700, 1 s)
    TagStructureMember "InWP"  LogicalAddress=%DB1020.DBX990.3
    TagStructureMember "InHP"  LogicalAddress=%DB1020.DBX990.4
    TagStructureMember "ValveType"  LogicalAddress=%DB1020.DBX990.5
    TagStructureMember "ManualToWP"  LogicalAddress=%DB1020.DBX996.0
    TagStructureMember "ManualToHP"  LogicalAddress=%DB1020.DBX996.1
    TagStructureMember "GoWorkTime"  LogicalAddress=%DB1020.DBW998
    TagStructureMember "GoHomeTime"  LogicalAddress=%DB1020.DBW1000
    TagStructureMember "oGoWP"  LogicalAddress=%DB1020.DBX1010.0
    TagStructureMember "oGoHP"  LogicalAddress=%DB1020.DBX1010.1
    TagStructureMember "oGoWPBTActive"  LogicalAddress=%DB1020.DBX1010.2
    TagStructureMember "oGoHPBTActive"  LogicalAddress=%DB1020.DBX1010.3
    TagStructureMember "CylinderNo"  LogicalAddress=%DB1020.DBB1011
  STxxxCylinder047 : fpCylinder V 0.0.19  (%DB1020.DBX1012.0, CPU S71500-2PN_TP700, 1 s)
    TagStructureMember "InWP"  LogicalAddress=%DB1020.DBX1012.3
    TagStructureMember "InHP"  LogicalAddress=%DB1020.DBX1012.4
    TagStructureMember "ValveType"  LogicalAddress=%DB1020.DBX1012.5
    TagStructureMember "ManualToWP"  LogicalAddress=%DB1020.DBX1018.0
    TagStructureMember "ManualToHP"  LogicalAddress=%DB1020.DBX1018.1
    TagStructureMember "GoWorkTime"  LogicalAddress=%DB1020.DBW1020
    TagStructureMember "GoHomeTime"  LogicalAddress=%DB1020.DBW1022
    TagStructureMember "oGoWP"  LogicalAddress=%DB1020.DBX1032.0
    TagStructureMember "oGoHP"  LogicalAddress=%DB1020.DBX1032.1
    TagStructureMember "oGoWPBTActive"  LogicalAddress=%DB1020.DBX1032.2
    TagStructureMember "oGoHPBTActive"  LogicalAddress=%DB1020.DBX1032.3
    TagStructureMember "CylinderNo"  LogicalAddress=%DB1020.DBB1033
  STxxxCylinder048 : fpCylinder V 0.0.19  (%DB1020.DBX1034.0, CPU S71500-2PN_TP700, 1 s)
    TagStructureMember "InWP"  LogicalAddress=%DB1020.DBX1034.3
    TagStructureMember "InHP"  LogicalAddress=%DB1020.DBX1034.4
    TagStructureMember "ValveType"  LogicalAddress=%DB1020.DBX1034.5
    TagStructureMember "ManualToWP"  LogicalAddress=%DB1020.DBX1040.0
    TagStructureMember "ManualToHP"  LogicalAddress=%DB1020.DBX1040.1
    TagStructureMember "GoWorkTime"  LogicalAddress=%DB1020.DBW1042
    TagStructureMember "GoHomeTime"  LogicalAddress=%DB1020.DBW1044
    TagStructureMember "oGoWP"  LogicalAddress=%DB1020.DBX1054.0
    TagStructureMember "oGoHP"  LogicalAddress=%DB1020.DBX1054.1
    TagStructureMember "oGoWPBTActive"  LogicalAddress=%DB1020.DBX1054.2
    TagStructureMember "oGoHPBTActive"  LogicalAddress=%DB1020.DBX1054.3
    TagStructureMember "CylinderNo"  LogicalAddress=%DB1020.DBB1055
  STxxxCylinder049 : fpCylinder V 0.0.19  (%DB1020.DBX1056.0, CPU S71500-2PN_TP700, 1 s)
    TagStructureMember "InWP"  LogicalAddress=%DB1020.DBX1056.3
    TagStructureMember "InHP"  LogicalAddress=%DB1020.DBX1056.4
    TagStructureMember "ValveType"  LogicalAddress=%DB1020.DBX1056.5
    TagStructureMember "ManualToWP"  LogicalAddress=%DB1020.DBX1062.0
    TagStructureMember "ManualToHP"  LogicalAddress=%DB1020.DBX1062.1
    TagStructureMember "GoWorkTime"  LogicalAddress=%DB1020.DBW1064
    TagStructureMember "GoHomeTime"  LogicalAddress=%DB1020.DBW1066
    TagStructureMember "oGoWP"  LogicalAddress=%DB1020.DBX1076.0
    TagStructureMember "oGoHP"  LogicalAddress=%DB1020.DBX1076.1
    TagStructureMember "oGoWPBTActive"  LogicalAddress=%DB1020.DBX1076.2
    TagStructureMember "oGoHPBTActive"  LogicalAddress=%DB1020.DBX1076.3
    TagStructureMember "CylinderNo"  LogicalAddress=%DB1020.DBB1077
  STxxxCylinder050 : fpCylinder V 0.0.19  (%DB1020.DBX1078.0, CPU S71500-2PN_TP700, 1 s)
    TagStructureMember "InWP"  LogicalAddress=%DB1020.DBX1078.3
    TagStructureMember "InHP"  LogicalAddress=%DB1020.DBX1078.4
    TagStructureMember "ValveType"  LogicalAddress=%DB1020.DBX1078.5
    TagStructureMember "ManualToWP"  LogicalAddress=%DB1020.DBX1084.0
    TagStructureMember "ManualToHP"  LogicalAddress=%DB1020.DBX1084.1
    TagStructureMember "GoWorkTime"  LogicalAddress=%DB1020.DBW1086
    TagStructureMember "GoHomeTime"  LogicalAddress=%DB1020.DBW1088
    TagStructureMember "oGoWP"  LogicalAddress=%DB1020.DBX1098.0
    TagStructureMember "oGoHP"  LogicalAddress=%DB1020.DBX1098.1
    TagStructureMember "oGoWPBTActive"  LogicalAddress=%DB1020.DBX1098.2
    TagStructureMember "oGoHPBTActive"  LogicalAddress=%DB1020.DBX1098.3
    TagStructureMember "CylinderNo"  LogicalAddress=%DB1020.DBB1099
  STxxxCylinder051 : fpCylinder V 0.0.19  (%DB1020.DBX1100.0, CPU S71500-2PN_TP700, 1 s)
    TagStructureMember "InWP"  LogicalAddress=%DB1020.DBX1100.3
    TagStructureMember "InHP"  LogicalAddress=%DB1020.DBX1100.4
    TagStructureMember "ValveType"  LogicalAddress=%DB1020.DBX1100.5
    TagStructureMember "ManualToWP"  LogicalAddress=%DB1020.DBX1106.0
    TagStructureMember "ManualToHP"  LogicalAddress=%DB1020.DBX1106.1
    TagStructureMember "GoWorkTime"  LogicalAddress=%DB1020.DBW1108
    TagStructureMember "GoHomeTime"  LogicalAddress=%DB1020.DBW1110
    TagStructureMember "oGoWP"  LogicalAddress=%DB1020.DBX1120.0
    TagStructureMember "oGoHP"  LogicalAddress=%DB1020.DBX1120.1
    TagStructureMember "oGoWPBTActive"  LogicalAddress=%DB1020.DBX1120.2
    TagStructureMember "oGoHPBTActive"  LogicalAddress=%DB1020.DBX1120.3
    TagStructureMember "CylinderNo"  LogicalAddress=%DB1020.DBB1121
  STxxxCylinder052 : fpCylinder V 0.0.19  (%DB1020.DBX1122.0, CPU S71500-2PN_TP700, 1 s)
    TagStructureMember "InWP"  LogicalAddress=%DB1020.DBX1122.3
    TagStructureMember "InHP"  LogicalAddress=%DB1020.DBX1122.4
    TagStructureMember "ValveType"  LogicalAddress=%DB1020.DBX1122.5
    TagStructureMember "ManualToWP"  LogicalAddress=%DB1020.DBX1128.0
    TagStructureMember "ManualToHP"  LogicalAddress=%DB1020.DBX1128.1
    TagStructureMember "GoWorkTime"  LogicalAddress=%DB1020.DBW1130
    TagStructureMember "GoHomeTime"  LogicalAddress=%DB1020.DBW1132
    TagStructureMember "oGoWP"  LogicalAddress=%DB1020.DBX1142.0
    TagStructureMember "oGoHP"  LogicalAddress=%DB1020.DBX1142.1
    TagStructureMember "oGoWPBTActive"  LogicalAddress=%DB1020.DBX1142.2
    TagStructureMember "oGoHPBTActive"  LogicalAddress=%DB1020.DBX1142.3
    TagStructureMember "CylinderNo"  LogicalAddress=%DB1020.DBB1143
  STxxxCylinder053 : fpCylinder V 0.0.19  (%DB1020.DBX1144.0, CPU S71500-2PN_TP700, 1 s)
    TagStructureMember "InWP"  LogicalAddress=%DB1020.DBX1144.3
    TagStructureMember "InHP"  LogicalAddress=%DB1020.DBX1144.4
    TagStructureMember "ValveType"  LogicalAddress=%DB1020.DBX1144.5
    TagStructureMember "ManualToWP"  LogicalAddress=%DB1020.DBX1150.0
    TagStructureMember "ManualToHP"  LogicalAddress=%DB1020.DBX1150.1
    TagStructureMember "GoWorkTime"  LogicalAddress=%DB1020.DBW1152
    TagStructureMember "GoHomeTime"  LogicalAddress=%DB1020.DBW1154
    TagStructureMember "oGoWP"  LogicalAddress=%DB1020.DBX1164.0
    TagStructureMember "oGoHP"  LogicalAddress=%DB1020.DBX1164.1
    TagStructureMember "oGoWPBTActive"  LogicalAddress=%DB1020.DBX1164.2
    TagStructureMember "oGoHPBTActive"  LogicalAddress=%DB1020.DBX1164.3
    TagStructureMember "CylinderNo"  LogicalAddress=%DB1020.DBB1165
  STxxxCylinder054 : fpCylinder V 0.0.19  (%DB1020.DBX1166.0, CPU S71500-2PN_TP700, 1 s)
    TagStructureMember "InWP"  LogicalAddress=%DB1020.DBX1166.3
    TagStructureMember "InHP"  LogicalAddress=%DB1020.DBX1166.4
    TagStructureMember "ValveType"  LogicalAddress=%DB1020.DBX1166.5
    TagStructureMember "ManualToWP"  LogicalAddress=%DB1020.DBX1172.0
    TagStructureMember "ManualToHP"  LogicalAddress=%DB1020.DBX1172.1
    TagStructureMember "GoWorkTime"  LogicalAddress=%DB1020.DBW1174
    TagStructureMember "GoHomeTime"  LogicalAddress=%DB1020.DBW1176
    TagStructureMember "oGoWP"  LogicalAddress=%DB1020.DBX1186.0
    TagStructureMember "oGoHP"  LogicalAddress=%DB1020.DBX1186.1
    TagStructureMember "oGoWPBTActive"  LogicalAddress=%DB1020.DBX1186.2
    TagStructureMember "oGoHPBTActive"  LogicalAddress=%DB1020.DBX1186.3
    TagStructureMember "CylinderNo"  LogicalAddress=%DB1020.DBB1187
  STxxxCylinder055 : fpCylinder V 0.0.19  (%DB1020.DBX1188.0, CPU S71500-2PN_TP700, 1 s)
    TagStructureMember "InWP"  LogicalAddress=%DB1020.DBX1188.3
    TagStructureMember "InHP"  LogicalAddress=%DB1020.DBX1188.4
    TagStructureMember "ValveType"  LogicalAddress=%DB1020.DBX1188.5
    TagStructureMember "ManualToWP"  LogicalAddress=%DB1020.DBX1194.0
    TagStructureMember "ManualToHP"  LogicalAddress=%DB1020.DBX1194.1
    TagStructureMember "GoWorkTime"  LogicalAddress=%DB1020.DBW1196
    TagStructureMember "GoHomeTime"  LogicalAddress=%DB1020.DBW1198
    TagStructureMember "oGoWP"  LogicalAddress=%DB1020.DBX1208.0
    TagStructureMember "oGoHP"  LogicalAddress=%DB1020.DBX1208.1
    TagStructureMember "oGoWPBTActive"  LogicalAddress=%DB1020.DBX1208.2
    TagStructureMember "oGoHPBTActive"  LogicalAddress=%DB1020.DBX1208.3
    TagStructureMember "CylinderNo"  LogicalAddress=%DB1020.DBB1209
  STxxxCylinder056 : fpCylinder V 0.0.19  (%DB1020.DBX1210.0, CPU S71500-2PN_TP700, 1 s)
    TagStructureMember "InWP"  LogicalAddress=%DB1020.DBX1210.3
    TagStructureMember "InHP"  LogicalAddress=%DB1020.DBX1210.4
    TagStructureMember "ValveType"  LogicalAddress=%DB1020.DBX1210.5
    TagStructureMember "ManualToWP"  LogicalAddress=%DB1020.DBX1216.0
    TagStructureMember "ManualToHP"  LogicalAddress=%DB1020.DBX1216.1
    TagStructureMember "GoWorkTime"  LogicalAddress=%DB1020.DBW1218
    TagStructureMember "GoHomeTime"  LogicalAddress=%DB1020.DBW1220
    TagStructureMember "oGoWP"  LogicalAddress=%DB1020.DBX1230.0
    TagStructureMember "oGoHP"  LogicalAddress=%DB1020.DBX1230.1
    TagStructureMember "oGoWPBTActive"  LogicalAddress=%DB1020.DBX1230.2
    TagStructureMember "oGoHPBTActive"  LogicalAddress=%DB1020.DBX1230.3
    TagStructureMember "CylinderNo"  LogicalAddress=%DB1020.DBB1231
  STxxxCylinder057 : fpCylinder V 0.0.19  (%DB1020.DBX1232.0, CPU S71500-2PN_TP700, 1 s)
    TagStructureMember "InWP"  LogicalAddress=%DB1020.DBX1232.3
    TagStructureMember "InHP"  LogicalAddress=%DB1020.DBX1232.4
    TagStructureMember "ValveType"  LogicalAddress=%DB1020.DBX1232.5
    TagStructureMember "ManualToWP"  LogicalAddress=%DB1020.DBX1238.0
    TagStructureMember "ManualToHP"  LogicalAddress=%DB1020.DBX1238.1
    TagStructureMember "GoWorkTime"  LogicalAddress=%DB1020.DBW1240
    TagStructureMember "GoHomeTime"  LogicalAddress=%DB1020.DBW1242
    TagStructureMember "oGoWP"  LogicalAddress=%DB1020.DBX1252.0
    TagStructureMember "oGoHP"  LogicalAddress=%DB1020.DBX1252.1
    TagStructureMember "oGoWPBTActive"  LogicalAddress=%DB1020.DBX1252.2
    TagStructureMember "oGoHPBTActive"  LogicalAddress=%DB1020.DBX1252.3
    TagStructureMember "CylinderNo"  LogicalAddress=%DB1020.DBB1253
  STxxxCylinder058 : fpCylinder V 0.0.19  (%DB1020.DBX1254.0, CPU S71500-2PN_TP700, 1 s)
    TagStructureMember "InWP"  LogicalAddress=%DB1020.DBX1254.3
    TagStructureMember "InHP"  LogicalAddress=%DB1020.DBX1254.4
    TagStructureMember "ValveType"  LogicalAddress=%DB1020.DBX1254.5
    TagStructureMember "ManualToWP"  LogicalAddress=%DB1020.DBX1260.0
    TagStructureMember "ManualToHP"  LogicalAddress=%DB1020.DBX1260.1
    TagStructureMember "GoWorkTime"  LogicalAddress=%DB1020.DBW1262
    TagStructureMember "GoHomeTime"  LogicalAddress=%DB1020.DBW1264
    TagStructureMember "oGoWP"  LogicalAddress=%DB1020.DBX1274.0
    TagStructureMember "oGoHP"  LogicalAddress=%DB1020.DBX1274.1
    TagStructureMember "oGoWPBTActive"  LogicalAddress=%DB1020.DBX1274.2
    TagStructureMember "oGoHPBTActive"  LogicalAddress=%DB1020.DBX1274.3
    TagStructureMember "CylinderNo"  LogicalAddress=%DB1020.DBB1275
  STxxxCylinder059 : fpCylinder V 0.0.19  (%DB1020.DBX1276.0, CPU S71500-2PN_TP700, 1 s)
    TagStructureMember "InWP"  LogicalAddress=%DB1020.DBX1276.3
    TagStructureMember "InHP"  LogicalAddress=%DB1020.DBX1276.4
    TagStructureMember "ValveType"  LogicalAddress=%DB1020.DBX1276.5
    TagStructureMember "ManualToWP"  LogicalAddress=%DB1020.DBX1282.0
    TagStructureMember "ManualToHP"  LogicalAddress=%DB1020.DBX1282.1
    TagStructureMember "GoWorkTime"  LogicalAddress=%DB1020.DBW1284
    TagStructureMember "GoHomeTime"  LogicalAddress=%DB1020.DBW1286
    TagStructureMember "oGoWP"  LogicalAddress=%DB1020.DBX1296.0
    TagStructureMember "oGoHP"  LogicalAddress=%DB1020.DBX1296.1
    TagStructureMember "oGoWPBTActive"  LogicalAddress=%DB1020.DBX1296.2
    TagStructureMember "oGoHPBTActive"  LogicalAddress=%DB1020.DBX1296.3
    TagStructureMember "CylinderNo"  LogicalAddress=%DB1020.DBB1297
  STxxxCylinder060 : fpCylinder V 0.0.19  (%DB1020.DBX1298.0, CPU S71500-2PN_TP700, 1 s)
    TagStructureMember "InWP"  LogicalAddress=%DB1020.DBX1298.3
    TagStructureMember "InHP"  LogicalAddress=%DB1020.DBX1298.4
    TagStructureMember "ValveType"  LogicalAddress=%DB1020.DBX1298.5
    TagStructureMember "ManualToWP"  LogicalAddress=%DB1020.DBX1304.0
    TagStructureMember "ManualToHP"  LogicalAddress=%DB1020.DBX1304.1
    TagStructureMember "GoWorkTime"  LogicalAddress=%DB1020.DBW1306
    TagStructureMember "GoHomeTime"  LogicalAddress=%DB1020.DBW1308
    TagStructureMember "oGoWP"  LogicalAddress=%DB1020.DBX1318.0
    TagStructureMember "oGoHP"  LogicalAddress=%DB1020.DBX1318.1
    TagStructureMember "oGoWPBTActive"  LogicalAddress=%DB1020.DBX1318.2
    TagStructureMember "oGoHPBTActive"  LogicalAddress=%DB1020.DBX1318.3
    TagStructureMember "CylinderNo"  LogicalAddress=%DB1020.DBB1319
  STxxxCylinder061 : fpCylinder V 0.0.19  (%DB1020.DBX1320.0, CPU S71500-2PN_TP700, 1 s)
    TagStructureMember "InWP"  LogicalAddress=%DB1020.DBX1320.3
    TagStructureMember "InHP"  LogicalAddress=%DB1020.DBX1320.4
    TagStructureMember "ValveType"  LogicalAddress=%DB1020.DBX1320.5
    TagStructureMember "ManualToWP"  LogicalAddress=%DB1020.DBX1326.0
    TagStructureMember "ManualToHP"  LogicalAddress=%DB1020.DBX1326.1
    TagStructureMember "GoWorkTime"  LogicalAddress=%DB1020.DBW1328
    TagStructureMember "GoHomeTime"  LogicalAddress=%DB1020.DBW1330
    TagStructureMember "oGoWP"  LogicalAddress=%DB1020.DBX1340.0
    TagStructureMember "oGoHP"  LogicalAddress=%DB1020.DBX1340.1
    TagStructureMember "oGoWPBTActive"  LogicalAddress=%DB1020.DBX1340.2
    TagStructureMember "oGoHPBTActive"  LogicalAddress=%DB1020.DBX1340.3
    TagStructureMember "CylinderNo"  LogicalAddress=%DB1020.DBB1341
  STxxxCylinder062 : fpCylinder V 0.0.19  (%DB1020.DBX1342.0, CPU S71500-2PN_TP700, 1 s)
    TagStructureMember "InWP"  LogicalAddress=%DB1020.DBX1342.3
    TagStructureMember "InHP"  LogicalAddress=%DB1020.DBX1342.4
    TagStructureMember "ValveType"  LogicalAddress=%DB1020.DBX1342.5
    TagStructureMember "ManualToWP"  LogicalAddress=%DB1020.DBX1348.0
    TagStructureMember "ManualToHP"  LogicalAddress=%DB1020.DBX1348.1
    TagStructureMember "GoWorkTime"  LogicalAddress=%DB1020.DBW1350
    TagStructureMember "GoHomeTime"  LogicalAddress=%DB1020.DBW1352
    TagStructureMember "oGoWP"  LogicalAddress=%DB1020.DBX1362.0
    TagStructureMember "oGoHP"  LogicalAddress=%DB1020.DBX1362.1
    TagStructureMember "oGoWPBTActive"  LogicalAddress=%DB1020.DBX1362.2
    TagStructureMember "oGoHPBTActive"  LogicalAddress=%DB1020.DBX1362.3
    TagStructureMember "CylinderNo"  LogicalAddress=%DB1020.DBB1363
  STxxxCylinder063 : fpCylinder V 0.0.19  (%DB1020.DBX1364.0, CPU S71500-2PN_TP700, 1 s)
    TagStructureMember "InWP"  LogicalAddress=%DB1020.DBX1364.3
    TagStructureMember "InHP"  LogicalAddress=%DB1020.DBX1364.4
    TagStructureMember "ValveType"  LogicalAddress=%DB1020.DBX1364.5
    TagStructureMember "ManualToWP"  LogicalAddress=%DB1020.DBX1370.0
    TagStructureMember "ManualToHP"  LogicalAddress=%DB1020.DBX1370.1
    TagStructureMember "GoWorkTime"  LogicalAddress=%DB1020.DBW1372
    TagStructureMember "GoHomeTime"  LogicalAddress=%DB1020.DBW1374
    TagStructureMember "oGoWP"  LogicalAddress=%DB1020.DBX1384.0
    TagStructureMember "oGoHP"  LogicalAddress=%DB1020.DBX1384.1
    TagStructureMember "oGoWPBTActive"  LogicalAddress=%DB1020.DBX1384.2
    TagStructureMember "oGoHPBTActive"  LogicalAddress=%DB1020.DBX1384.3
    TagStructureMember "CylinderNo"  LogicalAddress=%DB1020.DBB1385
  STxxxCylinder064 : fpCylinder V 0.0.19  (%DB1020.DBX1386.0, CPU S71500-2PN_TP700, 1 s)
    TagStructureMember "InWP"  LogicalAddress=%DB1020.DBX1386.3
    TagStructureMember "InHP"  LogicalAddress=%DB1020.DBX1386.4
    TagStructureMember "ValveType"  LogicalAddress=%DB1020.DBX1386.5
    TagStructureMember "ManualToWP"  LogicalAddress=%DB1020.DBX1392.0
    TagStructureMember "ManualToHP"  LogicalAddress=%DB1020.DBX1392.1
    TagStructureMember "GoWorkTime"  LogicalAddress=%DB1020.DBW1394
    TagStructureMember "GoHomeTime"  LogicalAddress=%DB1020.DBW1396
    TagStructureMember "oGoWP"  LogicalAddress=%DB1020.DBX1406.0
    TagStructureMember "oGoHP"  LogicalAddress=%DB1020.DBX1406.1
    TagStructureMember "oGoWPBTActive"  LogicalAddress=%DB1020.DBX1406.2
    TagStructureMember "oGoHPBTActive"  LogicalAddress=%DB1020.DBX1406.3
    TagStructureMember "CylinderNo"  LogicalAddress=%DB1020.DBB1407
  STxxxCylinder065 : fpCylinder V 0.0.19  (%DB1020.DBX1408.0, CPU S71500-2PN_TP700, 1 s)
    TagStructureMember "InWP"  LogicalAddress=%DB1020.DBX1408.3
    TagStructureMember "InHP"  LogicalAddress=%DB1020.DBX1408.4
    TagStructureMember "ValveType"  LogicalAddress=%DB1020.DBX1408.5
    TagStructureMember "ManualToWP"  LogicalAddress=%DB1020.DBX1414.0
    TagStructureMember "ManualToHP"  LogicalAddress=%DB1020.DBX1414.1
    TagStructureMember "GoWorkTime"  LogicalAddress=%DB1020.DBW1416
    TagStructureMember "GoHomeTime"  LogicalAddress=%DB1020.DBW1418
    TagStructureMember "oGoWP"  LogicalAddress=%DB1020.DBX1428.0
    TagStructureMember "oGoHP"  LogicalAddress=%DB1020.DBX1428.1
    TagStructureMember "oGoWPBTActive"  LogicalAddress=%DB1020.DBX1428.2
    TagStructureMember "oGoHPBTActive"  LogicalAddress=%DB1020.DBX1428.3
    TagStructureMember "CylinderNo"  LogicalAddress=%DB1020.DBB1429
  STxxxCylinder066 : fpCylinder V 0.0.19  (%DB1020.DBX1430.0, CPU S71500-2PN_TP700, 1 s)
    TagStructureMember "InWP"  LogicalAddress=%DB1020.DBX1430.3
    TagStructureMember "InHP"  LogicalAddress=%DB1020.DBX1430.4
    TagStructureMember "ValveType"  LogicalAddress=%DB1020.DBX1430.5
    TagStructureMember "ManualToWP"  LogicalAddress=%DB1020.DBX1436.0
    TagStructureMember "ManualToHP"  LogicalAddress=%DB1020.DBX1436.1
    TagStructureMember "GoWorkTime"  LogicalAddress=%DB1020.DBW1438
    TagStructureMember "GoHomeTime"  LogicalAddress=%DB1020.DBW1440
    TagStructureMember "oGoWP"  LogicalAddress=%DB1020.DBX1450.0
    TagStructureMember "oGoHP"  LogicalAddress=%DB1020.DBX1450.1
    TagStructureMember "oGoWPBTActive"  LogicalAddress=%DB1020.DBX1450.2
    TagStructureMember "oGoHPBTActive"  LogicalAddress=%DB1020.DBX1450.3
    TagStructureMember "CylinderNo"  LogicalAddress=%DB1020.DBB1451
  STxxxCylinder067 : fpCylinder V 0.0.19  (%DB1020.DBX1452.0, CPU S71500-2PN_TP700, 1 s)
    TagStructureMember "InWP"  LogicalAddress=%DB1020.DBX1452.3
    TagStructureMember "InHP"  LogicalAddress=%DB1020.DBX1452.4
    TagStructureMember "ValveType"  LogicalAddress=%DB1020.DBX1452.5
    TagStructureMember "ManualToWP"  LogicalAddress=%DB1020.DBX1458.0
    TagStructureMember "ManualToHP"  LogicalAddress=%DB1020.DBX1458.1
    TagStructureMember "GoWorkTime"  LogicalAddress=%DB1020.DBW1460
    TagStructureMember "GoHomeTime"  LogicalAddress=%DB1020.DBW1462
    TagStructureMember "oGoWP"  LogicalAddress=%DB1020.DBX1472.0
    TagStructureMember "oGoHP"  LogicalAddress=%DB1020.DBX1472.1
    TagStructureMember "oGoWPBTActive"  LogicalAddress=%DB1020.DBX1472.2
    TagStructureMember "oGoHPBTActive"  LogicalAddress=%DB1020.DBX1472.3
    TagStructureMember "CylinderNo"  LogicalAddress=%DB1020.DBB1473
  STxxxCylinder068 : fpCylinder V 0.0.19  (%DB1020.DBX1474.0, CPU S71500-2PN_TP700, 1 s)
    TagStructureMember "InWP"  LogicalAddress=%DB1020.DBX1474.3
    TagStructureMember "InHP"  LogicalAddress=%DB1020.DBX1474.4
    TagStructureMember "ValveType"  LogicalAddress=%DB1020.DBX1474.5
    TagStructureMember "ManualToWP"  LogicalAddress=%DB1020.DBX1480.0
    TagStructureMember "ManualToHP"  LogicalAddress=%DB1020.DBX1480.1
    TagStructureMember "GoWorkTime"  LogicalAddress=%DB1020.DBW1482
    TagStructureMember "GoHomeTime"  LogicalAddress=%DB1020.DBW1484
    TagStructureMember "oGoWP"  LogicalAddress=%DB1020.DBX1494.0
    TagStructureMember "oGoHP"  LogicalAddress=%DB1020.DBX1494.1
    TagStructureMember "oGoWPBTActive"  LogicalAddress=%DB1020.DBX1494.2
    TagStructureMember "oGoHPBTActive"  LogicalAddress=%DB1020.DBX1494.3
    TagStructureMember "CylinderNo"  LogicalAddress=%DB1020.DBB1495
  STxxxCylinder069 : fpCylinder V 0.0.19  (%DB1020.DBX1496.0, CPU S71500-2PN_TP700, 1 s)
    TagStructureMember "InWP"  LogicalAddress=%DB1020.DBX1496.3
    TagStructureMember "InHP"  LogicalAddress=%DB1020.DBX1496.4
    TagStructureMember "ValveType"  LogicalAddress=%DB1020.DBX1496.5
    TagStructureMember "ManualToWP"  LogicalAddress=%DB1020.DBX1502.0
    TagStructureMember "ManualToHP"  LogicalAddress=%DB1020.DBX1502.1
    TagStructureMember "GoWorkTime"  LogicalAddress=%DB1020.DBW1504
    TagStructureMember "GoHomeTime"  LogicalAddress=%DB1020.DBW1506
    TagStructureMember "oGoWP"  LogicalAddress=%DB1020.DBX1516.0
    TagStructureMember "oGoHP"  LogicalAddress=%DB1020.DBX1516.1
    TagStructureMember "oGoWPBTActive"  LogicalAddress=%DB1020.DBX1516.2
    TagStructureMember "oGoHPBTActive"  LogicalAddress=%DB1020.DBX1516.3
    TagStructureMember "CylinderNo"  LogicalAddress=%DB1020.DBB1517
  STxxxCylinder070 : fpCylinder V 0.0.19  (%DB1020.DBX1518.0, CPU S71500-2PN_TP700, 1 s)
    TagStructureMember "InWP"  LogicalAddress=%DB1020.DBX1518.3
    TagStructureMember "InHP"  LogicalAddress=%DB1020.DBX1518.4
    TagStructureMember "ValveType"  LogicalAddress=%DB1020.DBX1518.5
    TagStructureMember "ManualToWP"  LogicalAddress=%DB1020.DBX1524.0
    TagStructureMember "ManualToHP"  LogicalAddress=%DB1020.DBX1524.1
    TagStructureMember "GoWorkTime"  LogicalAddress=%DB1020.DBW1526
    TagStructureMember "GoHomeTime"  LogicalAddress=%DB1020.DBW1528
    TagStructureMember "oGoWP"  LogicalAddress=%DB1020.DBX1538.0
    TagStructureMember "oGoHP"  LogicalAddress=%DB1020.DBX1538.1
    TagStructureMember "oGoWPBTActive"  LogicalAddress=%DB1020.DBX1538.2
    TagStructureMember "oGoHPBTActive"  LogicalAddress=%DB1020.DBX1538.3
    TagStructureMember "CylinderNo"  LogicalAddress=%DB1020.DBB1539
  STxxxCylinder071 : fpCylinder V 0.0.19  (%DB1020.DBX1540.0, CPU S71500-2PN_TP700, 1 s)
    TagStructureMember "InWP"  LogicalAddress=%DB1020.DBX1540.3
    TagStructureMember "InHP"  LogicalAddress=%DB1020.DBX1540.4
    TagStructureMember "ValveType"  LogicalAddress=%DB1020.DBX1540.5
    TagStructureMember "ManualToWP"  LogicalAddress=%DB1020.DBX1546.0
    TagStructureMember "ManualToHP"  LogicalAddress=%DB1020.DBX1546.1
    TagStructureMember "GoWorkTime"  LogicalAddress=%DB1020.DBW1548
    TagStructureMember "GoHomeTime"  LogicalAddress=%DB1020.DBW1550
    TagStructureMember "oGoWP"  LogicalAddress=%DB1020.DBX1560.0
    TagStructureMember "oGoHP"  LogicalAddress=%DB1020.DBX1560.1
    TagStructureMember "oGoWPBTActive"  LogicalAddress=%DB1020.DBX1560.2
    TagStructureMember "oGoHPBTActive"  LogicalAddress=%DB1020.DBX1560.3
    TagStructureMember "CylinderNo"  LogicalAddress=%DB1020.DBB1561
  STxxxCylinder072 : fpCylinder V 0.0.19  (%DB1020.DBX1562.0, CPU S71500-2PN_TP700, 1 s)
    TagStructureMember "InWP"  LogicalAddress=%DB1020.DBX1562.3
    TagStructureMember "InHP"  LogicalAddress=%DB1020.DBX1562.4
    TagStructureMember "ValveType"  LogicalAddress=%DB1020.DBX1562.5
    TagStructureMember "ManualToWP"  LogicalAddress=%DB1020.DBX1568.0
    TagStructureMember "ManualToHP"  LogicalAddress=%DB1020.DBX1568.1
    TagStructureMember "GoWorkTime"  LogicalAddress=%DB1020.DBW1570
    TagStructureMember "GoHomeTime"  LogicalAddress=%DB1020.DBW1572
    TagStructureMember "oGoWP"  LogicalAddress=%DB1020.DBX1582.0
    TagStructureMember "oGoHP"  LogicalAddress=%DB1020.DBX1582.1
    TagStructureMember "oGoWPBTActive"  LogicalAddress=%DB1020.DBX1582.2
    TagStructureMember "oGoHPBTActive"  LogicalAddress=%DB1020.DBX1582.3
    TagStructureMember "CylinderNo"  LogicalAddress=%DB1020.DBB1583
  STxxxCylinder073 : fpCylinder V 0.0.19  (%DB1020.DBX1584.0, CPU S71500-2PN_TP700, 1 s)
    TagStructureMember "InWP"  LogicalAddress=%DB1020.DBX1584.3
    TagStructureMember "InHP"  LogicalAddress=%DB1020.DBX1584.4
    TagStructureMember "ValveType"  LogicalAddress=%DB1020.DBX1584.5
    TagStructureMember "ManualToWP"  LogicalAddress=%DB1020.DBX1590.0
    TagStructureMember "ManualToHP"  LogicalAddress=%DB1020.DBX1590.1
    TagStructureMember "GoWorkTime"  LogicalAddress=%DB1020.DBW1592
    TagStructureMember "GoHomeTime"  LogicalAddress=%DB1020.DBW1594
    TagStructureMember "oGoWP"  LogicalAddress=%DB1020.DBX1604.0
    TagStructureMember "oGoHP"  LogicalAddress=%DB1020.DBX1604.1
    TagStructureMember "oGoWPBTActive"  LogicalAddress=%DB1020.DBX1604.2
    TagStructureMember "oGoHPBTActive"  LogicalAddress=%DB1020.DBX1604.3
    TagStructureMember "CylinderNo"  LogicalAddress=%DB1020.DBB1605
  STxxxCylinder074 : fpCylinder V 0.0.19  (%DB1020.DBX1606.0, CPU S71500-2PN_TP700, 1 s)
    TagStructureMember "InWP"  LogicalAddress=%DB1020.DBX1606.3
    TagStructureMember "InHP"  LogicalAddress=%DB1020.DBX1606.4
    TagStructureMember "ValveType"  LogicalAddress=%DB1020.DBX1606.5
    TagStructureMember "ManualToWP"  LogicalAddress=%DB1020.DBX1612.0
    TagStructureMember "ManualToHP"  LogicalAddress=%DB1020.DBX1612.1
    TagStructureMember "GoWorkTime"  LogicalAddress=%DB1020.DBW1614
    TagStructureMember "GoHomeTime"  LogicalAddress=%DB1020.DBW1616
    TagStructureMember "oGoWP"  LogicalAddress=%DB1020.DBX1626.0
    TagStructureMember "oGoHP"  LogicalAddress=%DB1020.DBX1626.1
    TagStructureMember "oGoWPBTActive"  LogicalAddress=%DB1020.DBX1626.2
    TagStructureMember "oGoHPBTActive"  LogicalAddress=%DB1020.DBX1626.3
    TagStructureMember "CylinderNo"  LogicalAddress=%DB1020.DBB1627
  STxxxCylinder075 : fpCylinder V 0.0.19  (%DB1020.DBX1628.0, CPU S71500-2PN_TP700, 1 s)
    TagStructureMember "InWP"  LogicalAddress=%DB1020.DBX1628.3
    TagStructureMember "InHP"  LogicalAddress=%DB1020.DBX1628.4
    TagStructureMember "ValveType"  LogicalAddress=%DB1020.DBX1628.5
    TagStructureMember "ManualToWP"  LogicalAddress=%DB1020.DBX1634.0
    TagStructureMember "ManualToHP"  LogicalAddress=%DB1020.DBX1634.1
    TagStructureMember "GoWorkTime"  LogicalAddress=%DB1020.DBW1636
    TagStructureMember "GoHomeTime"  LogicalAddress=%DB1020.DBW1638
    TagStructureMember "oGoWP"  LogicalAddress=%DB1020.DBX1648.0
    TagStructureMember "oGoHP"  LogicalAddress=%DB1020.DBX1648.1
    TagStructureMember "oGoWPBTActive"  LogicalAddress=%DB1020.DBX1648.2
    TagStructureMember "oGoHPBTActive"  LogicalAddress=%DB1020.DBX1648.3
    TagStructureMember "CylinderNo"  LogicalAddress=%DB1020.DBB1649
  STxxxCylinder076 : fpCylinder V 0.0.19  (%DB1020.DBX1650.0, CPU S71500-2PN_TP700, 1 s)
    TagStructureMember "InWP"  LogicalAddress=%DB1020.DBX1650.3
    TagStructureMember "InHP"  LogicalAddress=%DB1020.DBX1650.4
    TagStructureMember "ValveType"  LogicalAddress=%DB1020.DBX1650.5
    TagStructureMember "ManualToWP"  LogicalAddress=%DB1020.DBX1656.0
    TagStructureMember "ManualToHP"  LogicalAddress=%DB1020.DBX1656.1
    TagStructureMember "GoWorkTime"  LogicalAddress=%DB1020.DBW1658
    TagStructureMember "GoHomeTime"  LogicalAddress=%DB1020.DBW1660
    TagStructureMember "oGoWP"  LogicalAddress=%DB1020.DBX1670.0
    TagStructureMember "oGoHP"  LogicalAddress=%DB1020.DBX1670.1
    TagStructureMember "oGoWPBTActive"  LogicalAddress=%DB1020.DBX1670.2
    TagStructureMember "oGoHPBTActive"  LogicalAddress=%DB1020.DBX1670.3
    TagStructureMember "CylinderNo"  LogicalAddress=%DB1020.DBB1671
  STxxxCylinder077 : fpCylinder V 0.0.19  (%DB1020.DBX1672.0, CPU S71500-2PN_TP700, 1 s)
    TagStructureMember "InWP"  LogicalAddress=%DB1020.DBX1672.3
    TagStructureMember "InHP"  LogicalAddress=%DB1020.DBX1672.4
    TagStructureMember "ValveType"  LogicalAddress=%DB1020.DBX1672.5
    TagStructureMember "ManualToWP"  LogicalAddress=%DB1020.DBX1678.0
    TagStructureMember "ManualToHP"  LogicalAddress=%DB1020.DBX1678.1
    TagStructureMember "GoWorkTime"  LogicalAddress=%DB1020.DBW1680
    TagStructureMember "GoHomeTime"  LogicalAddress=%DB1020.DBW1682
    TagStructureMember "oGoWP"  LogicalAddress=%DB1020.DBX1692.0
    TagStructureMember "oGoHP"  LogicalAddress=%DB1020.DBX1692.1
    TagStructureMember "oGoWPBTActive"  LogicalAddress=%DB1020.DBX1692.2
    TagStructureMember "oGoHPBTActive"  LogicalAddress=%DB1020.DBX1692.3
    TagStructureMember "CylinderNo"  LogicalAddress=%DB1020.DBB1693
  STxxxCylinder078 : fpCylinder V 0.0.19  (%DB1020.DBX1694.0, CPU S71500-2PN_TP700, 1 s)
    TagStructureMember "InWP"  LogicalAddress=%DB1020.DBX1694.3
    TagStructureMember "InHP"  LogicalAddress=%DB1020.DBX1694.4
    TagStructureMember "ValveType"  LogicalAddress=%DB1020.DBX1694.5
    TagStructureMember "ManualToWP"  LogicalAddress=%DB1020.DBX1700.0
    TagStructureMember "ManualToHP"  LogicalAddress=%DB1020.DBX1700.1
    TagStructureMember "GoWorkTime"  LogicalAddress=%DB1020.DBW1702
    TagStructureMember "GoHomeTime"  LogicalAddress=%DB1020.DBW1704
    TagStructureMember "oGoWP"  LogicalAddress=%DB1020.DBX1714.0
    TagStructureMember "oGoHP"  LogicalAddress=%DB1020.DBX1714.1
    TagStructureMember "oGoWPBTActive"  LogicalAddress=%DB1020.DBX1714.2
    TagStructureMember "oGoHPBTActive"  LogicalAddress=%DB1020.DBX1714.3
    TagStructureMember "CylinderNo"  LogicalAddress=%DB1020.DBB1715
  STxxxCylinder079 : fpCylinder V 0.0.19  (%DB1020.DBX1716.0, CPU S71500-2PN_TP700, 1 s)
    TagStructureMember "InWP"  LogicalAddress=%DB1020.DBX1716.3
    TagStructureMember "InHP"  LogicalAddress=%DB1020.DBX1716.4
    TagStructureMember "ValveType"  LogicalAddress=%DB1020.DBX1716.5
    TagStructureMember "ManualToWP"  LogicalAddress=%DB1020.DBX1722.0
    TagStructureMember "ManualToHP"  LogicalAddress=%DB1020.DBX1722.1
    TagStructureMember "GoWorkTime"  LogicalAddress=%DB1020.DBW1724
    TagStructureMember "GoHomeTime"  LogicalAddress=%DB1020.DBW1726
    TagStructureMember "oGoWP"  LogicalAddress=%DB1020.DBX1736.0
    TagStructureMember "oGoHP"  LogicalAddress=%DB1020.DBX1736.1
    TagStructureMember "oGoWPBTActive"  LogicalAddress=%DB1020.DBX1736.2
    TagStructureMember "oGoHPBTActive"  LogicalAddress=%DB1020.DBX1736.3
    TagStructureMember "CylinderNo"  LogicalAddress=%DB1020.DBB1737
  STxxxCylinder080 : fpCylinder V 0.0.19  (%DB1020.DBX1738.0, CPU S71500-2PN_TP700, 1 s)
    TagStructureMember "InWP"  LogicalAddress=%DB1020.DBX1738.3
    TagStructureMember "InHP"  LogicalAddress=%DB1020.DBX1738.4
    TagStructureMember "ValveType"  LogicalAddress=%DB1020.DBX1738.5
    TagStructureMember "ManualToWP"  LogicalAddress=%DB1020.DBX1744.0
    TagStructureMember "ManualToHP"  LogicalAddress=%DB1020.DBX1744.1
    TagStructureMember "GoWorkTime"  LogicalAddress=%DB1020.DBW1746
    TagStructureMember "GoHomeTime"  LogicalAddress=%DB1020.DBW1748
    TagStructureMember "oGoWP"  LogicalAddress=%DB1020.DBX1758.0
    TagStructureMember "oGoHP"  LogicalAddress=%DB1020.DBX1758.1
    TagStructureMember "oGoWPBTActive"  LogicalAddress=%DB1020.DBX1758.2
    TagStructureMember "oGoHPBTActive"  LogicalAddress=%DB1020.DBX1758.3
    TagStructureMember "CylinderNo"  LogicalAddress=%DB1020.DBB1759
  STxxxCylinder081 : fpCylinder V 0.0.19  (%DB1020.DBX1760.0, CPU S71500-2PN_TP700, 1 s)
    TagStructureMember "InWP"  LogicalAddress=%DB1020.DBX1760.3
    TagStructureMember "InHP"  LogicalAddress=%DB1020.DBX1760.4
    TagStructureMember "ValveType"  LogicalAddress=%DB1020.DBX1760.5
    TagStructureMember "ManualToWP"  LogicalAddress=%DB1020.DBX1766.0
    TagStructureMember "ManualToHP"  LogicalAddress=%DB1020.DBX1766.1
    TagStructureMember "GoWorkTime"  LogicalAddress=%DB1020.DBW1768
    TagStructureMember "GoHomeTime"  LogicalAddress=%DB1020.DBW1770
    TagStructureMember "oGoWP"  LogicalAddress=%DB1020.DBX1780.0
    TagStructureMember "oGoHP"  LogicalAddress=%DB1020.DBX1780.1
    TagStructureMember "oGoWPBTActive"  LogicalAddress=%DB1020.DBX1780.2
    TagStructureMember "oGoHPBTActive"  LogicalAddress=%DB1020.DBX1780.3
    TagStructureMember "CylinderNo"  LogicalAddress=%DB1020.DBB1781
  STxxxCylinder082 : fpCylinder V 0.0.19  (%DB1020.DBX1782.0, CPU S71500-2PN_TP700, 1 s)
    TagStructureMember "InWP"  LogicalAddress=%DB1020.DBX1782.3
    TagStructureMember "InHP"  LogicalAddress=%DB1020.DBX1782.4
    TagStructureMember "ValveType"  LogicalAddress=%DB1020.DBX1782.5
    TagStructureMember "ManualToWP"  LogicalAddress=%DB1020.DBX1788.0
    TagStructureMember "ManualToHP"  LogicalAddress=%DB1020.DBX1788.1
    TagStructureMember "GoWorkTime"  LogicalAddress=%DB1020.DBW1790
    TagStructureMember "GoHomeTime"  LogicalAddress=%DB1020.DBW1792
    TagStructureMember "oGoWP"  LogicalAddress=%DB1020.DBX1802.0
    TagStructureMember "oGoHP"  LogicalAddress=%DB1020.DBX1802.1
    TagStructureMember "oGoWPBTActive"  LogicalAddress=%DB1020.DBX1802.2
    TagStructureMember "oGoHPBTActive"  LogicalAddress=%DB1020.DBX1802.3
    TagStructureMember "CylinderNo"  LogicalAddress=%DB1020.DBB1803
  STxxxCylinder083 : fpCylinder V 0.0.19  (%DB1020.DBX1804.0, CPU S71500-2PN_TP700, 1 s)
    TagStructureMember "InWP"  LogicalAddress=%DB1020.DBX1804.3
    TagStructureMember "InHP"  LogicalAddress=%DB1020.DBX1804.4
    TagStructureMember "ValveType"  LogicalAddress=%DB1020.DBX1804.5
    TagStructureMember "ManualToWP"  LogicalAddress=%DB1020.DBX1810.0
    TagStructureMember "ManualToHP"  LogicalAddress=%DB1020.DBX1810.1
    TagStructureMember "GoWorkTime"  LogicalAddress=%DB1020.DBW1812
    TagStructureMember "GoHomeTime"  LogicalAddress=%DB1020.DBW1814
    TagStructureMember "oGoWP"  LogicalAddress=%DB1020.DBX1824.0
    TagStructureMember "oGoHP"  LogicalAddress=%DB1020.DBX1824.1
    TagStructureMember "oGoWPBTActive"  LogicalAddress=%DB1020.DBX1824.2
    TagStructureMember "oGoHPBTActive"  LogicalAddress=%DB1020.DBX1824.3
    TagStructureMember "CylinderNo"  LogicalAddress=%DB1020.DBB1825
  STxxxCylinder084 : fpCylinder V 0.0.19  (%DB1020.DBX1826.0, CPU S71500-2PN_TP700, 1 s)
    TagStructureMember "InWP"  LogicalAddress=%DB1020.DBX1826.3
    TagStructureMember "InHP"  LogicalAddress=%DB1020.DBX1826.4
    TagStructureMember "ValveType"  LogicalAddress=%DB1020.DBX1826.5
    TagStructureMember "ManualToWP"  LogicalAddress=%DB1020.DBX1832.0
    TagStructureMember "ManualToHP"  LogicalAddress=%DB1020.DBX1832.1
    TagStructureMember "GoWorkTime"  LogicalAddress=%DB1020.DBW1834
    TagStructureMember "GoHomeTime"  LogicalAddress=%DB1020.DBW1836
    TagStructureMember "oGoWP"  LogicalAddress=%DB1020.DBX1846.0
    TagStructureMember "oGoHP"  LogicalAddress=%DB1020.DBX1846.1
    TagStructureMember "oGoWPBTActive"  LogicalAddress=%DB1020.DBX1846.2
    TagStructureMember "oGoHPBTActive"  LogicalAddress=%DB1020.DBX1846.3
    TagStructureMember "CylinderNo"  LogicalAddress=%DB1020.DBB1847
  STxxxCylinder085 : fpCylinder V 0.0.19  (%DB1020.DBX1848.0, CPU S71500-2PN_TP700, 1 s)
    TagStructureMember "InWP"  LogicalAddress=%DB1020.DBX1848.3
    TagStructureMember "InHP"  LogicalAddress=%DB1020.DBX1848.4
    TagStructureMember "ValveType"  LogicalAddress=%DB1020.DBX1848.5
    TagStructureMember "ManualToWP"  LogicalAddress=%DB1020.DBX1854.0
    TagStructureMember "ManualToHP"  LogicalAddress=%DB1020.DBX1854.1
    TagStructureMember "GoWorkTime"  LogicalAddress=%DB1020.DBW1856
    TagStructureMember "GoHomeTime"  LogicalAddress=%DB1020.DBW1858
    TagStructureMember "oGoWP"  LogicalAddress=%DB1020.DBX1868.0
    TagStructureMember "oGoHP"  LogicalAddress=%DB1020.DBX1868.1
    TagStructureMember "oGoWPBTActive"  LogicalAddress=%DB1020.DBX1868.2
    TagStructureMember "oGoHPBTActive"  LogicalAddress=%DB1020.DBX1868.3
    TagStructureMember "CylinderNo"  LogicalAddress=%DB1020.DBB1869
  STxxxCylinder086 : fpCylinder V 0.0.19  (%DB1020.DBX1870.0, CPU S71500-2PN_TP700, 1 s)
    TagStructureMember "InWP"  LogicalAddress=%DB1020.DBX1870.3
    TagStructureMember "InHP"  LogicalAddress=%DB1020.DBX1870.4
    TagStructureMember "ValveType"  LogicalAddress=%DB1020.DBX1870.5
    TagStructureMember "ManualToWP"  LogicalAddress=%DB1020.DBX1876.0
    TagStructureMember "ManualToHP"  LogicalAddress=%DB1020.DBX1876.1
    TagStructureMember "GoWorkTime"  LogicalAddress=%DB1020.DBW1878
    TagStructureMember "GoHomeTime"  LogicalAddress=%DB1020.DBW1880
    TagStructureMember "oGoWP"  LogicalAddress=%DB1020.DBX1890.0
    TagStructureMember "oGoHP"  LogicalAddress=%DB1020.DBX1890.1
    TagStructureMember "oGoWPBTActive"  LogicalAddress=%DB1020.DBX1890.2
    TagStructureMember "oGoHPBTActive"  LogicalAddress=%DB1020.DBX1890.3
    TagStructureMember "CylinderNo"  LogicalAddress=%DB1020.DBB1891
  STxxxCylinder087 : fpCylinder V 0.0.19  (%DB1020.DBX1892.0, CPU S71500-2PN_TP700, 1 s)
    TagStructureMember "InWP"  LogicalAddress=%DB1020.DBX1892.3
    TagStructureMember "InHP"  LogicalAddress=%DB1020.DBX1892.4
    TagStructureMember "ValveType"  LogicalAddress=%DB1020.DBX1892.5
    TagStructureMember "ManualToWP"  LogicalAddress=%DB1020.DBX1898.0
    TagStructureMember "ManualToHP"  LogicalAddress=%DB1020.DBX1898.1
    TagStructureMember "GoWorkTime"  LogicalAddress=%DB1020.DBW1900
    TagStructureMember "GoHomeTime"  LogicalAddress=%DB1020.DBW1902
    TagStructureMember "oGoWP"  LogicalAddress=%DB1020.DBX1912.0
    TagStructureMember "oGoHP"  LogicalAddress=%DB1020.DBX1912.1
    TagStructureMember "oGoWPBTActive"  LogicalAddress=%DB1020.DBX1912.2
    TagStructureMember "oGoHPBTActive"  LogicalAddress=%DB1020.DBX1912.3
    TagStructureMember "CylinderNo"  LogicalAddress=%DB1020.DBB1913
  STxxxCylinder088 : fpCylinder V 0.0.19  (%DB1020.DBX1914.0, CPU S71500-2PN_TP700, 1 s)
    TagStructureMember "InWP"  LogicalAddress=%DB1020.DBX1914.3
    TagStructureMember "InHP"  LogicalAddress=%DB1020.DBX1914.4
    TagStructureMember "ValveType"  LogicalAddress=%DB1020.DBX1914.5
    TagStructureMember "ManualToWP"  LogicalAddress=%DB1020.DBX1920.0
    TagStructureMember "ManualToHP"  LogicalAddress=%DB1020.DBX1920.1
    TagStructureMember "GoWorkTime"  LogicalAddress=%DB1020.DBW1922
    TagStructureMember "GoHomeTime"  LogicalAddress=%DB1020.DBW1924
    TagStructureMember "oGoWP"  LogicalAddress=%DB1020.DBX1934.0
    TagStructureMember "oGoHP"  LogicalAddress=%DB1020.DBX1934.1
    TagStructureMember "oGoWPBTActive"  LogicalAddress=%DB1020.DBX1934.2
    TagStructureMember "oGoHPBTActive"  LogicalAddress=%DB1020.DBX1934.3
    TagStructureMember "CylinderNo"  LogicalAddress=%DB1020.DBB1935
  STxxxCylinder089 : fpCylinder V 0.0.19  (%DB1020.DBX1936.0, CPU S71500-2PN_TP700, 1 s)
    TagStructureMember "InWP"  LogicalAddress=%DB1020.DBX1936.3
    TagStructureMember "InHP"  LogicalAddress=%DB1020.DBX1936.4
    TagStructureMember "ValveType"  LogicalAddress=%DB1020.DBX1936.5
    TagStructureMember "ManualToWP"  LogicalAddress=%DB1020.DBX1942.0
    TagStructureMember "ManualToHP"  LogicalAddress=%DB1020.DBX1942.1
    TagStructureMember "GoWorkTime"  LogicalAddress=%DB1020.DBW1944
    TagStructureMember "GoHomeTime"  LogicalAddress=%DB1020.DBW1946
    TagStructureMember "oGoWP"  LogicalAddress=%DB1020.DBX1956.0
    TagStructureMember "oGoHP"  LogicalAddress=%DB1020.DBX1956.1
    TagStructureMember "oGoWPBTActive"  LogicalAddress=%DB1020.DBX1956.2
    TagStructureMember "oGoHPBTActive"  LogicalAddress=%DB1020.DBX1956.3
    TagStructureMember "CylinderNo"  LogicalAddress=%DB1020.DBB1957
  STxxxCylinder090 : fpCylinder V 0.0.19  (%DB1020.DBX1958.0, CPU S71500-2PN_TP700, 1 s)
    TagStructureMember "InWP"  LogicalAddress=%DB1020.DBX1958.3
    TagStructureMember "InHP"  LogicalAddress=%DB1020.DBX1958.4
    TagStructureMember "ValveType"  LogicalAddress=%DB1020.DBX1958.5
    TagStructureMember "ManualToWP"  LogicalAddress=%DB1020.DBX1964.0
    TagStructureMember "ManualToHP"  LogicalAddress=%DB1020.DBX1964.1
    TagStructureMember "GoWorkTime"  LogicalAddress=%DB1020.DBW1966
    TagStructureMember "GoHomeTime"  LogicalAddress=%DB1020.DBW1968
    TagStructureMember "oGoWP"  LogicalAddress=%DB1020.DBX1978.0
    TagStructureMember "oGoHP"  LogicalAddress=%DB1020.DBX1978.1
    TagStructureMember "oGoWPBTActive"  LogicalAddress=%DB1020.DBX1978.2
    TagStructureMember "oGoHPBTActive"  LogicalAddress=%DB1020.DBX1978.3
    TagStructureMember "CylinderNo"  LogicalAddress=%DB1020.DBB1979
  STxxxCylinder091 : fpCylinder V 0.0.19  (%DB1020.DBX1980.0, CPU S71500-2PN_TP700, 1 s)
    TagStructureMember "InWP"  LogicalAddress=%DB1020.DBX1980.3
    TagStructureMember "InHP"  LogicalAddress=%DB1020.DBX1980.4
    TagStructureMember "ValveType"  LogicalAddress=%DB1020.DBX1980.5
    TagStructureMember "ManualToWP"  LogicalAddress=%DB1020.DBX1986.0
    TagStructureMember "ManualToHP"  LogicalAddress=%DB1020.DBX1986.1
    TagStructureMember "GoWorkTime"  LogicalAddress=%DB1020.DBW1988
    TagStructureMember "GoHomeTime"  LogicalAddress=%DB1020.DBW1990
    TagStructureMember "oGoWP"  LogicalAddress=%DB1020.DBX2000.0
    TagStructureMember "oGoHP"  LogicalAddress=%DB1020.DBX2000.1
    TagStructureMember "oGoWPBTActive"  LogicalAddress=%DB1020.DBX2000.2
    TagStructureMember "oGoHPBTActive"  LogicalAddress=%DB1020.DBX2000.3
    TagStructureMember "CylinderNo"  LogicalAddress=%DB1020.DBB2001
  STxxxCylinder092 : fpCylinder V 0.0.19  (%DB1020.DBX2002.0, CPU S71500-2PN_TP700, 1 s)
    TagStructureMember "InWP"  LogicalAddress=%DB1020.DBX2002.3
    TagStructureMember "InHP"  LogicalAddress=%DB1020.DBX2002.4
    TagStructureMember "ValveType"  LogicalAddress=%DB1020.DBX2002.5
    TagStructureMember "ManualToWP"  LogicalAddress=%DB1020.DBX2008.0
    TagStructureMember "ManualToHP"  LogicalAddress=%DB1020.DBX2008.1
    TagStructureMember "GoWorkTime"  LogicalAddress=%DB1020.DBW2010
    TagStructureMember "GoHomeTime"  LogicalAddress=%DB1020.DBW2012
    TagStructureMember "oGoWP"  LogicalAddress=%DB1020.DBX2022.0
    TagStructureMember "oGoHP"  LogicalAddress=%DB1020.DBX2022.1
    TagStructureMember "oGoWPBTActive"  LogicalAddress=%DB1020.DBX2022.2
    TagStructureMember "oGoHPBTActive"  LogicalAddress=%DB1020.DBX2022.3
    TagStructureMember "CylinderNo"  LogicalAddress=%DB1020.DBB2023
  STxxxCylinder093 : fpCylinder V 0.0.19  (%DB1020.DBX2024.0, CPU S71500-2PN_TP700, 1 s)
    TagStructureMember "InWP"  LogicalAddress=%DB1020.DBX2024.3
    TagStructureMember "InHP"  LogicalAddress=%DB1020.DBX2024.4
    TagStructureMember "ValveType"  LogicalAddress=%DB1020.DBX2024.5
    TagStructureMember "ManualToWP"  LogicalAddress=%DB1020.DBX2030.0
    TagStructureMember "ManualToHP"  LogicalAddress=%DB1020.DBX2030.1
    TagStructureMember "GoWorkTime"  LogicalAddress=%DB1020.DBW2032
    TagStructureMember "GoHomeTime"  LogicalAddress=%DB1020.DBW2034
    TagStructureMember "oGoWP"  LogicalAddress=%DB1020.DBX2044.0
    TagStructureMember "oGoHP"  LogicalAddress=%DB1020.DBX2044.1
    TagStructureMember "oGoWPBTActive"  LogicalAddress=%DB1020.DBX2044.2
    TagStructureMember "oGoHPBTActive"  LogicalAddress=%DB1020.DBX2044.3
    TagStructureMember "CylinderNo"  LogicalAddress=%DB1020.DBB2045
  STxxxCylinder094 : fpCylinder V 0.0.19  (%DB1020.DBX2046.0, CPU S71500-2PN_TP700, 1 s)
    TagStructureMember "InWP"  LogicalAddress=%DB1020.DBX2046.3
    TagStructureMember "InHP"  LogicalAddress=%DB1020.DBX2046.4
    TagStructureMember "ValveType"  LogicalAddress=%DB1020.DBX2046.5
    TagStructureMember "ManualToWP"  LogicalAddress=%DB1020.DBX2052.0
    TagStructureMember "ManualToHP"  LogicalAddress=%DB1020.DBX2052.1
    TagStructureMember "GoWorkTime"  LogicalAddress=%DB1020.DBW2054
    TagStructureMember "GoHomeTime"  LogicalAddress=%DB1020.DBW2056
    TagStructureMember "oGoWP"  LogicalAddress=%DB1020.DBX2066.0
    TagStructureMember "oGoHP"  LogicalAddress=%DB1020.DBX2066.1
    TagStructureMember "oGoWPBTActive"  LogicalAddress=%DB1020.DBX2066.2
    TagStructureMember "oGoHPBTActive"  LogicalAddress=%DB1020.DBX2066.3
    TagStructureMember "CylinderNo"  LogicalAddress=%DB1020.DBB2067
  STxxxCylinder095 : fpCylinder V 0.0.19  (%DB1020.DBX2068.0, CPU S71500-2PN_TP700, 1 s)
    TagStructureMember "InWP"  LogicalAddress=%DB1020.DBX2068.3
    TagStructureMember "InHP"  LogicalAddress=%DB1020.DBX2068.4
    TagStructureMember "ValveType"  LogicalAddress=%DB1020.DBX2068.5
    TagStructureMember "ManualToWP"  LogicalAddress=%DB1020.DBX2074.0
    TagStructureMember "ManualToHP"  LogicalAddress=%DB1020.DBX2074.1
    TagStructureMember "GoWorkTime"  LogicalAddress=%DB1020.DBW2076
    TagStructureMember "GoHomeTime"  LogicalAddress=%DB1020.DBW2078
    TagStructureMember "oGoWP"  LogicalAddress=%DB1020.DBX2088.0
    TagStructureMember "oGoHP"  LogicalAddress=%DB1020.DBX2088.1
    TagStructureMember "oGoWPBTActive"  LogicalAddress=%DB1020.DBX2088.2
    TagStructureMember "oGoHPBTActive"  LogicalAddress=%DB1020.DBX2088.3
    TagStructureMember "CylinderNo"  LogicalAddress=%DB1020.DBB2089
  STxxxCylinder096 : fpCylinder V 0.0.19  (%DB1020.DBX2090.0, CPU S71500-2PN_TP700, 1 s)
    TagStructureMember "InWP"  LogicalAddress=%DB1020.DBX2090.3
    TagStructureMember "InHP"  LogicalAddress=%DB1020.DBX2090.4
    TagStructureMember "ValveType"  LogicalAddress=%DB1020.DBX2090.5
    TagStructureMember "ManualToWP"  LogicalAddress=%DB1020.DBX2096.0
    TagStructureMember "ManualToHP"  LogicalAddress=%DB1020.DBX2096.1
    TagStructureMember "GoWorkTime"  LogicalAddress=%DB1020.DBW2098
    TagStructureMember "GoHomeTime"  LogicalAddress=%DB1020.DBW2100
    TagStructureMember "oGoWP"  LogicalAddress=%DB1020.DBX2110.0
    TagStructureMember "oGoHP"  LogicalAddress=%DB1020.DBX2110.1
    TagStructureMember "oGoWPBTActive"  LogicalAddress=%DB1020.DBX2110.2
    TagStructureMember "oGoHPBTActive"  LogicalAddress=%DB1020.DBX2110.3
    TagStructureMember "CylinderNo"  LogicalAddress=%DB1020.DBB2111
  STxxxCylinder097 : fpCylinder V 0.0.19  (%DB1020.DBX2112.0, CPU S71500-2PN_TP700, 1 s)
    TagStructureMember "InWP"  LogicalAddress=%DB1020.DBX2112.3
    TagStructureMember "InHP"  LogicalAddress=%DB1020.DBX2112.4
    TagStructureMember "ValveType"  LogicalAddress=%DB1020.DBX2112.5
    TagStructureMember "ManualToWP"  LogicalAddress=%DB1020.DBX2118.0
    TagStructureMember "ManualToHP"  LogicalAddress=%DB1020.DBX2118.1
    TagStructureMember "GoWorkTime"  LogicalAddress=%DB1020.DBW2120
    TagStructureMember "GoHomeTime"  LogicalAddress=%DB1020.DBW2122
    TagStructureMember "oGoWP"  LogicalAddress=%DB1020.DBX2132.0
    TagStructureMember "oGoHP"  LogicalAddress=%DB1020.DBX2132.1
    TagStructureMember "oGoWPBTActive"  LogicalAddress=%DB1020.DBX2132.2
    TagStructureMember "oGoHPBTActive"  LogicalAddress=%DB1020.DBX2132.3
    TagStructureMember "CylinderNo"  LogicalAddress=%DB1020.DBB2133
  STxxxCylinder098 : fpCylinder V 0.0.19  (%DB1020.DBX2134.0, CPU S71500-2PN_TP700, 1 s)
    TagStructureMember "InWP"  LogicalAddress=%DB1020.DBX2134.3
    TagStructureMember "InHP"  LogicalAddress=%DB1020.DBX2134.4
    TagStructureMember "ValveType"  LogicalAddress=%DB1020.DBX2134.5
    TagStructureMember "ManualToWP"  LogicalAddress=%DB1020.DBX2140.0
    TagStructureMember "ManualToHP"  LogicalAddress=%DB1020.DBX2140.1
    TagStructureMember "GoWorkTime"  LogicalAddress=%DB1020.DBW2142
    TagStructureMember "GoHomeTime"  LogicalAddress=%DB1020.DBW2144
    TagStructureMember "oGoWP"  LogicalAddress=%DB1020.DBX2154.0
    TagStructureMember "oGoHP"  LogicalAddress=%DB1020.DBX2154.1
    TagStructureMember "oGoWPBTActive"  LogicalAddress=%DB1020.DBX2154.2
    TagStructureMember "oGoHPBTActive"  LogicalAddress=%DB1020.DBX2154.3
    TagStructureMember "CylinderNo"  LogicalAddress=%DB1020.DBB2155
  STxxxCylinder099 : fpCylinder V 0.0.19  (%DB1020.DBX2156.0, CPU S71500-2PN_TP700, 1 s)
    TagStructureMember "InWP"  LogicalAddress=%DB1020.DBX2156.3
    TagStructureMember "InHP"  LogicalAddress=%DB1020.DBX2156.4
    TagStructureMember "ValveType"  LogicalAddress=%DB1020.DBX2156.5
    TagStructureMember "ManualToWP"  LogicalAddress=%DB1020.DBX2162.0
    TagStructureMember "ManualToHP"  LogicalAddress=%DB1020.DBX2162.1
    TagStructureMember "GoWorkTime"  LogicalAddress=%DB1020.DBW2164
    TagStructureMember "GoHomeTime"  LogicalAddress=%DB1020.DBW2166
    TagStructureMember "oGoWP"  LogicalAddress=%DB1020.DBX2176.0
    TagStructureMember "oGoHP"  LogicalAddress=%DB1020.DBX2176.1
    TagStructureMember "oGoWPBTActive"  LogicalAddress=%DB1020.DBX2176.2
    TagStructureMember "oGoHPBTActive"  LogicalAddress=%DB1020.DBX2176.3
    TagStructureMember "CylinderNo"  LogicalAddress=%DB1020.DBB2177
  STxxxCylinder100 : fpCylinder V 0.0.19  (%DB1020.DBX2178.0, CPU S71500-2PN_TP700, 1 s)
    TagStructureMember "InWP"  LogicalAddress=%DB1020.DBX2178.3
    TagStructureMember "InHP"  LogicalAddress=%DB1020.DBX2178.4
    TagStructureMember "ValveType"  LogicalAddress=%DB1020.DBX2178.5
    TagStructureMember "ManualToWP"  LogicalAddress=%DB1020.DBX2184.0
    TagStructureMember "ManualToHP"  LogicalAddress=%DB1020.DBX2184.1
    TagStructureMember "GoWorkTime"  LogicalAddress=%DB1020.DBW2186
    TagStructureMember "GoHomeTime"  LogicalAddress=%DB1020.DBW2188
    TagStructureMember "oGoWP"  LogicalAddress=%DB1020.DBX2198.0
    TagStructureMember "oGoHP"  LogicalAddress=%DB1020.DBX2198.1
    TagStructureMember "oGoWPBTActive"  LogicalAddress=%DB1020.DBX2198.2
    TagStructureMember "oGoHPBTActive"  LogicalAddress=%DB1020.DBX2198.3
    TagStructureMember "CylinderNo"  LogicalAddress=%DB1020.DBB2199
